LIN {X 0,Y 373.398,Z 423.906,A -85,B 0,C 180,E1 -12851.054,E2 -12851.054} C_VEL
LIN {X 0,Y 371.737,Z 434.746,A -85,B 0,C 180,E1 -12852.96,E2 -12852.96} C_VEL
LIN {X 0,Y 370.406,Z 443.745,A -85,B 0,C 180,E1 -12854.877,E2 -12854.877} C_VEL
LIN {X 0,Y 369.476,Z 451.202,A -85,B 0,C 180,E1 -12856.805,E2 -12856.805} C_VEL
LIN {X 0,Y 368.494,Z 458.177,A -85,B 0,C 180,E1 -12859.005,E2 -12859.005} C_VEL
LIN {X 0,Y 367.969,Z 463.658,A -85,B 0,C 180,E1 -12861.211,E2 -12861.211} C_VEL
LIN {X 0,Y 367.613,Z 468.407,A -85,B 0,C 180,E1 -12863.791,E2 -12863.791} C_VEL
LIN {X 0,Y 367.456,Z 470.707,A -85,B 0,C 180,E1 -12865.612,E2 -12865.612} C_VEL
LIN {X 0,Y 367.353,Z 472.458,A -85,B 0,C 180,E1 -12867.807,E2 -12867.807} C_VEL
LIN {X 0,Y 367.373,Z 473.069,A -85,B 0,C 180,E1 -12870,E2 -12870} C_VEL
LIN {X 0,Y 367.353,Z 472.504,A -85,B 0,C 180,E1 -12872.193,E2 -12872.193} C_VEL
LIN {X 0,Y 367.45,Z 470.815,A -85,B 0,C 180,E1 -12874.388,E2 -12874.388} C_VEL
LIN {X 0,Y 367.559,Z 467.963,A -85,B 0,C 180,E1 -12876.588,E2 -12876.588} C_VEL
LIN {X 0,Y 367.957,Z 463.881,A -85,B 0,C 180,E1 -12878.789,E2 -12878.789} C_VEL
LIN {X 0,Y 368.468,Z 458.469,A -85,B 0,C 180,E1 -12880.996,E2 -12880.996} C_VEL
LIN {X 0,Y 368.933,Z 455.452,A -85,B 0,C 180,E1 -12882.017,E2 -12882.017} C_VEL
LIN {X 0,Y 368.664,Z 452.923,A -85,B 0,C 180,E1 -12882.844,E2 -12882.844} C_VEL
LIN {X 0,Y 366.408,Z 448.547,A -85,B 0,C 180,E1 -12884.185,E2 -12884.185} C_VEL
LIN {X 0,Y 364.21,Z 443.754,A -85,B 0,C 180,E1 -12885.503,E2 -12885.503} C_VEL
LIN {X 0,Y 364.039,Z 440.47,A -85,B 0,C 180,E1 -12886.282,E2 -12886.282} C_VEL
LIN {X 0,Y 365.526,Z 430.926,A -85,B 0,C 180,E1 -12888.206,E2 -12888.206} C_VEL
LIN {X 0,Y 367.184,Z 421.057,A -85,B 0,C 180,E1 -12889.861,E2 -12889.861} C_VEL
LIN {X 0,Y 368.721,Z 410.391,A -85,B 0,C 180,E1 -12891.379,E2 -12891.379} C_VEL
LIN {X 0,Y 370.415,Z 398.934,A -85,B 0,C 180,E1 -12892.742,E2 -12892.742} C_VEL
LIN {X 0,Y 372.09,Z 386.634,A -85,B 0,C 180,E1 -12893.96,E2 -12893.96} C_VEL
LIN {X 0,Y 373.712,Z 373.285,A -85,B 0,C 180,E1 -12895.033,E2 -12895.033} C_VEL
LIN {X 0,Y 375.189,Z 358.112,A -85,B 0,C 180,E1 -12895.993,E2 -12895.993} C_VEL
LIN {X 0,Y 376.337,Z 343.059,A -85,B 0,C 180,E1 -12896.703,E2 -12896.703} C_VEL
LIN {X 0,Y 377.198,Z 327.711,A -85,B 0,C 180,E1 -12897.198,E2 -12897.198} C_VEL
LIN {X 0,Y 380.187,Z 211.478,A -85,B 0,C 180,E1 -12899.438,E2 -12899.438} C_VEL
LIN {X 0,Y 380.388,Z 200.049,A -85,B 0,C 180,E1 -12899.664,E2 -12899.664} C_VEL
LIN {X 0,Y 378.985,Z 193.552,A -85,B 0,C 180,E1 -12899.924,E2 -12899.924} C_VEL
LIN {X 0,Y 370.925,Z 175.178,A -85,B 0,C 180,E1 -12901.05,E2 -12901.05} C_VEL
LIN {X 0,Y 364.955,Z 162.744,A -85,B 0,C 180,E1 -12901.927,E2 -12901.927} C_VEL
LIN {X 0,Y 362.572,Z 153.728,A -85,B 0,C 180,E1 -12904.203,E2 -12904.203} C_VEL
LIN {X 0,Y 361.902,Z 151.154,A -85,B 0,C 180,E1 -12904.951,E2 -12904.951} C_VEL
LIN {X 0,Y 361.843,Z 151.036,A -85,B 0,C 180,E1 -12908.428,E2 -12908.428} C_VEL
LIN {X 0,Y 361.823,Z 151.038,A -85,B 0,C 180,E1 -12912.429,E2 -12912.429} C_VEL
LIN {X 0,Y 361.814,Z 151.039,A -85,B 0,C 180,E1 -12915.948,E2 -12915.948} C_VEL
LIN {X 0,Y 361.81,Z 151.006,A -85,B 0,C 180,E1 -12919.25,E2 -12919.25} C_VEL
LIN {X 0,Y 361.865,Z 151.034,A -85,B 0,C 180,E1 -12922.982,E2 -12922.982} C_VEL
LIN {X 0,Y 361.859,Z 150.996,A -85,B 0,C 180,E1 -12926.631,E2 -12926.631} C_VEL
LIN {X 0,Y 361.849,Z 151.006,A -85,B 0,C 180,E1 -12929.67,E2 -12929.67} C_VEL
LIN {X 0,Y 361.863,Z 151.032,A -85,B 0,C 180,E1 -12933.468,E2 -12933.468} C_VEL
LIN {X 0,Y 361.877,Z 151.031,A -85,B 0,C 180,E1 -12937.144,E2 -12937.144} C_VEL
LIN {X 0,Y 361.885,Z 151.02,A -85,B 0,C 180,E1 -12940.722,E2 -12940.722} C_VEL
LIN {X 0,Y 361.907,Z 151.02,A -85,B 0,C 180,E1 -12944.224,E2 -12944.224} C_VEL
LIN {X 0,Y 362.001,Z 151.007,A -85,B 0,C 180,E1 -12946.528,E2 -12946.528} C_VEL
LIN {X 0,Y 362.002,Z 151.01,A -85,B 0,C 180,E1 -12949.937,E2 -12949.937} C_VEL
LIN {X 0,Y 362.141,Z 150.993,A -85,B 0,C 180,E1 -12953.313,E2 -12953.313} C_VEL
LIN {X 0,Y 362.27,Z 150.965,A -85,B 0,C 180,E1 -12957.776,E2 -12957.776} C_VEL
LIN {X 0,Y 362.382,Z 150.968,A -85,B 0,C 180,E1 -12960,E2 -12960} C_VEL
LIN {X 0,Y 362.274,Z 150.973,A -85,B 0,C 180,E1 -12962.223,E2 -12962.223} C_VEL
LIN {X 0,Y 362.137,Z 150.998,A -85,B 0,C 180,E1 -12966.687,E2 -12966.687} C_VEL
LIN {X 0,Y 362.002,Z 151.001,A -85,B 0,C 180,E1 -12970.063,E2 -12970.063} C_VEL
LIN {X 0,Y 362,Z 151.012,A -85,B 0,C 180,E1 -12973.899,E2 -12973.899} C_VEL
LIN {X 0,Y 361.969,Z 151.02,A -85,B 0,C 180,E1 -12977.938,E2 -12977.938} C_VEL
LIN {X 0,Y 361.862,Z 151.024,A -85,B 0,C 180,E1 -12981.655,E2 -12981.655} C_VEL
LIN {X 0,Y 361.927,Z 151.015,A -85,B 0,C 180,E1 -12985.29,E2 -12985.29} C_VEL
LIN {X 0,Y 361.919,Z 151.025,A -85,B 0,C 180,E1 -12987.778,E2 -12987.778} C_VEL
LIN {X 0,Y 361.847,Z 151.006,A -85,B 0,C 180,E1 -12991.285,E2 -12991.285} C_VEL
LIN {X 0,Y 361.854,Z 150.999,A -85,B 0,C 180,E1 -12994.28,E2 -12994.28} C_VEL
LIN {X 0,Y 361.864,Z 151.034,A -85,B 0,C 180,E1 -12997.223,E2 -12997.223} C_VEL
LIN {X 0,Y 361.835,Z 151.007,A -85,B 0,C 180,E1 -13000.755,E2 -13000.755} C_VEL
LIN {X 0,Y 361.818,Z 151.034,A -85,B 0,C 180,E1 -13004.368,E2 -13004.368} C_VEL
LIN {X 0,Y 361.836,Z 151.03,A -85,B 0,C 180,E1 -13007.568,E2 -13007.568} C_VEL
LIN {X 0,Y 361.869,Z 151.018,A -85,B 0,C 180,E1 -13010.973,E2 -13010.973} C_VEL
LIN {X 0,Y 361.911,Z 151.209,A -85,B 0,C 180,E1 -13013.982,E2 -13013.982} C_VEL
LIN {X 0,Y 365.189,Z 163.283,A -85,B 0,C 180,E1 -13017.076,E2 -13017.076} C_VEL
LIN {X 0,Y 366.498,Z 168.406,A -85,B 0,C 180,E1 -13018.267,E2 -13018.267} C_VEL
LIN {X 0,Y 375.255,Z 187.677,A -85,B 0,C 180,E1 -13019.533,E2 -13019.533} C_VEL
LIN {X 0,Y 377.161,Z 192.668,A -85,B 0,C 180,E1 -13019.811,E2 -13019.811} C_VEL
LIN {X 0,Y 380.221,Z 208.628,A -85,B 0,C 180,E1 -13020.418,E2 -13020.418} C_VEL
LIN {X 0,Y 377.778,Z 309.972,A -85,B 0,C 180,E1 -13022.359,E2 -13022.359} C_VEL
LIN {X 0,Y 377.001,Z 336.104,A -85,B 0,C 180,E1 -13022.899,E2 -13022.899} C_VEL
LIN {X 0,Y 376.013,Z 351.534,A -85,B 0,C 180,E1 -13023.422,E2 -13023.422} C_VEL
LIN {X 0,Y 374.858,Z 365.308,A -85,B 0,C 180,E1 -13024.083,E2 -13024.083} C_VEL
LIN {X 0,Y 373.48,Z 379.072,A -85,B 0,C 180,E1 -13024.953,E2 -13024.953} C_VEL
LIN {X 0,Y 371.868,Z 392.508,A -85,B 0,C 180,E1 -13026.025,E2 -13026.025} C_VEL
LIN {X 0,Y 370.134,Z 404.922,A -85,B 0,C 180,E1 -13027.24,E2 -13027.24} C_VEL
LIN {X 0,Y 368.423,Z 416.478,A -85,B 0,C 180,E1 -13028.603,E2 -13028.603} C_VEL
LIN {X 0,Y 366.803,Z 427.233,A -85,B 0,C 180,E1 -13030.117,E2 -13030.117} C_VEL
LIN {X 0,Y 365.213,Z 437.183,A -85,B 0,C 180,E1 -13031.777,E2 -13031.777} C_VEL
LIN {X 0,Y 363.743,Z 446.916,A -85,B 0,C 180,E1 -13033.73,E2 -13033.73} C_VEL
LIN {X 0,Y 362.496,Z 455.382,A -85,B 0,C 180,E1 -13035.786,E2 -13035.786} C_VEL
LIN {X 0,Y 361.752,Z 461.749,A -85,B 0,C 180,E1 -13037.66,E2 -13037.66} C_VEL
LIN {X 0,Y 360.971,Z 467.946,A -85,B 0,C 180,E1 -13039.908,E2 -13039.908} C_VEL
LIN {X 0,Y 360.582,Z 472.739,A -85,B 0,C 180,E1 -13042.158,E2 -13042.158} C_VEL
LIN {X 0,Y 360.344,Z 476.249,A -85,B 0,C 180,E1 -13044.404,E2 -13044.404} C_VEL
LIN {X 0,Y 360.256,Z 478.558,A -85,B 0,C 180,E1 -13046.645,E2 -13046.645} C_VEL
LIN {X 0,Y 360.245,Z 479.718,A -85,B 0,C 180,E1 -13048.882,E2 -13048.882} C_VEL
LIN {X 0,Y 360.245,Z 479.716,A -85,B 0,C 180,E1 -13051.118,E2 -13051.118} C_VEL
LIN {X 0,Y 360.256,Z 478.546,A -85,B 0,C 180,E1 -13053.355,E2 -13053.355} C_VEL
LIN {X 0,Y 360.348,Z 476.23,A -85,B 0,C 180,E1 -13055.596,E2 -13055.596} C_VEL
LIN {X 0,Y 360.592,Z 472.718,A -85,B 0,C 180,E1 -13057.841,E2 -13057.841} C_VEL
LIN {X 0,Y 360.967,Z 467.92,A -85,B 0,C 180,E1 -13060.092,E2 -13060.092} C_VEL
LIN {X 0,Y 361.746,Z 461.706,A -85,B 0,C 180,E1 -13062.34,E2 -13062.34} C_VEL
LIN {X 0,Y 362.669,Z 453.9,A -85,B 0,C 180,E1 -13064.591,E2 -13064.591} C_VEL
LIN {X 0,Y 363.927,Z 445.6,A -85,B 0,C 180,E1 -13066.55,E2 -13066.55} C_VEL
LIN {X 0,Y 365.473,Z 435.597,A -85,B 0,C 180,E1 -13068.499,E2 -13068.499} C_VEL
LIN {X 0,Y 367.05,Z 424.826,A -85,B 0,C 180,E1 -13070.246,E2 -13070.246} C_VEL
LIN {X 0,Y 368.909,Z 413.17,A -85,B 0,C 180,E1 -13071.808,E2 -13071.808} C_VEL
LIN {X 0,Y 370.812,Z 399.587,A -85,B 0,C 180,E1 -13073.306,E2 -13073.306} C_VEL
LIN {X 0,Y 372.652,Z 385.966,A -85,B 0,C 180,E1 -13074.514,E2 -13074.514} C_VEL
LIN {X 0,Y 374.206,Z 371.977,A -85,B 0,C 180,E1 -13075.509,E2 -13075.509} C_VEL
LIN {X 0,Y 375.479,Z 357.981,A -85,B 0,C 180,E1 -13076.282,E2 -13076.282} C_VEL
LIN {X 0,Y 376.618,Z 342.393,A -85,B 0,C 180,E1 -13076.906,E2 -13076.906} C_VEL
LIN {X 0,Y 377.293,Z 327.061,A -85,B 0,C 180,E1 -13077.303,E2 -13077.303} C_VEL
LIN {X 0,Y 380.19,Z 209.703,A -85,B 0,C 180,E1 -13079.545,E2 -13079.545} C_VEL
LIN {X 0,Y 377.93,Z 196.695,A -85,B 0,C 180,E1 -13080.018,E2 -13080.018} C_VEL
LIN {X 0,Y 376.432,Z 190.399,A -85,B 0,C 180,E1 -13080.285,E2 -13080.285} C_VEL
LIN {X 0,Y 368.092,Z 171.918,A -85,B 0,C 180,E1 -13081.457,E2 -13081.457} C_VEL
LIN {X 0,Y 366.407,Z 168.152,A -85,B 0,C 180,E1 -13081.753,E2 -13081.753} C_VEL
LIN {X 0,Y 363.562,Z 157.181,A -85,B 0,C 180,E1 -13084.432,E2 -13084.432} C_VEL
LIN {X 0,Y 361.894,Z 151.108,A -85,B 0,C 180,E1 -13086.063,E2 -13086.063} C_VEL
LIN {X 0,Y 361.854,Z 151.019,A -85,B 0,C 180,E1 -13089.861,E2 -13089.861} C_VEL
LIN {X 0,Y 361.836,Z 151.022,A -85,B 0,C 180,E1 -13092.829,E2 -13092.829} C_VEL
LIN {X 0,Y 361.819,Z 151.039,A -85,B 0,C 180,E1 -13095.947,E2 -13095.947} C_VEL
LIN {X 0,Y 361.835,Z 151.007,A -85,B 0,C 180,E1 -13099.245,E2 -13099.245} C_VEL
LIN {X 0,Y 361.863,Z 151.034,A -85,B 0,C 180,E1 -13102.777,E2 -13102.777} C_VEL
LIN {X 0,Y 361.853,Z 150.998,A -85,B 0,C 180,E1 -13105.72,E2 -13105.72} C_VEL
LIN {X 0,Y 361.875,Z 151.019,A -85,B 0,C 180,E1 -13109.672,E2 -13109.672} C_VEL
LIN {X 0,Y 361.955,Z 151.01,A -85,B 0,C 180,E1 -13113.475,E2 -13113.475} C_VEL
LIN {X 0,Y 361.891,Z 151.028,A -85,B 0,C 180,E1 -13117.145,E2 -13117.145} C_VEL
LIN {X 0,Y 361.907,Z 151.025,A -85,B 0,C 180,E1 -13120.724,E2 -13120.724} C_VEL
LIN {X 0,Y 361.934,Z 151.018,A -85,B 0,C 180,E1 -13123.066,E2 -13123.066} C_VEL
LIN {X 0,Y 362,Z 151.014,A -85,B 0,C 180,E1 -13126.528,E2 -13126.528} C_VEL
LIN {X 0,Y 362.001,Z 151.001,A -85,B 0,C 180,E1 -13129.937,E2 -13129.937} C_VEL
LIN {X 0,Y 362.137,Z 150.998,A -85,B 0,C 180,E1 -13133.313,E2 -13133.313} C_VEL
LIN {X 0,Y 362.279,Z 150.972,A -85,B 0,C 180,E1 -13137.777,E2 -13137.777} C_VEL
LIN {X 0,Y 362.403,Z 150.965,A -85,B 0,C 180,E1 -13140,E2 -13140} C_VEL
LIN {X 0,Y 362.271,Z 150.965,A -85,B 0,C 180,E1 -13142.224,E2 -13142.224} C_VEL
LIN {X 0,Y 362.141,Z 150.994,A -85,B 0,C 180,E1 -13146.687,E2 -13146.687} C_VEL
LIN {X 0,Y 362.001,Z 151.009,A -85,B 0,C 180,E1 -13150.063,E2 -13150.063} C_VEL
LIN {X 0,Y 362,Z 151.003,A -85,B 0,C 180,E1 -13153.899,E2 -13153.899} C_VEL
LIN {X 0,Y 361.928,Z 151.025,A -85,B 0,C 180,E1 -13156.934,E2 -13156.934} C_VEL
LIN {X 0,Y 361.887,Z 151.018,A -85,B 0,C 180,E1 -13160.461,E2 -13160.461} C_VEL
LIN {X 0,Y 361.862,Z 151.026,A -85,B 0,C 180,E1 -13164.101,E2 -13164.101} C_VEL
LIN {X 0,Y 361.841,Z 151.04,A -85,B 0,C 180,E1 -13167.785,E2 -13167.785} C_VEL
LIN {X 0,Y 361.846,Z 150.992,A -85,B 0,C 180,E1 -13171.285,E2 -13171.285} C_VEL
LIN {X 0,Y 361.854,Z 151.011,A -85,B 0,C 180,E1 -13174.281,E2 -13174.281} C_VEL
LIN {X 0,Y 361.861,Z 151.033,A -85,B 0,C 180,E1 -13177.222,E2 -13177.222} C_VEL
LIN {X 0,Y 361.812,Z 151.003,A -85,B 0,C 180,E1 -13180.751,E2 -13180.751} C_VEL
LIN {X 0,Y 361.815,Z 151.038,A -85,B 0,C 180,E1 -13184.369,E2 -13184.369} C_VEL
LIN {X 0,Y 361.826,Z 151.035,A -85,B 0,C 180,E1 -13187.57,E2 -13187.57} C_VEL
LIN {X 0,Y 361.844,Z 151.034,A -85,B 0,C 180,E1 -13191.572,E2 -13191.572} C_VEL
LIN {X 0,Y 361.921,Z 151.113,A -85,B 0,C 180,E1 -13195.136,E2 -13195.136} C_VEL
LIN {X 0,Y 362.737,Z 154.31,A -85,B 0,C 180,E1 -13196.064,E2 -13196.064} C_VEL
LIN {X 0,Y 365.002,Z 162.815,A -85,B 0,C 180,E1 -13198.195,E2 -13198.195} C_VEL
LIN {X 0,Y 374.821,Z 183.627,A -85,B 0,C 180,E1 -13199.6,E2 -13199.6} C_VEL
LIN {X 0,Y 379.252,Z 194.366,A -85,B 0,C 180,E1 -13200.224,E2 -13200.224} C_VEL
LIN {X 0,Y 380.41,Z 201.067,A -85,B 0,C 180,E1 -13200.466,E2 -13200.466} C_VEL
LIN {X 0,Y 377.588,Z 313.354,A -85,B 0,C 180,E1 -13202.607,E2 -13202.607} C_VEL
LIN {X 0,Y 376.944,Z 332.564,A -85,B 0,C 180,E1 -13203.044,E2 -13203.044} C_VEL
LIN {X 0,Y 375.949,Z 347.72,A -85,B 0,C 180,E1 -13203.598,E2 -13203.598} C_VEL
LIN {X 0,Y 374.794,Z 362.411,A -85,B 0,C 180,E1 -13204.363,E2 -13204.363} C_VEL
LIN {X 0,Y 373.413,Z 375.563,A -85,B 0,C 180,E1 -13205.243,E2 -13205.243} C_VEL
LIN {X 0,Y 371.763,Z 388.509,A -85,B 0,C 180,E1 -13206.314,E2 -13206.314} C_VEL
LIN {X 0,Y 369.97,Z 401.744,A -85,B 0,C 180,E1 -13207.671,E2 -13207.671} C_VEL
LIN {X 0,Y 368.388,Z 412.361,A -85,B 0,C 180,E1 -13208.975,E2 -13208.975} C_VEL
LIN {X 0,Y 366.673,Z 423.976,A -85,B 0,C 180,E1 -13210.693,E2 -13210.693} C_VEL
LIN {X 0,Y 364.905,Z 434.816,A -85,B 0,C 180,E1 -13212.631,E2 -13212.631} C_VEL
LIN {X 0,Y 363.485,Z 443.814,A -85,B 0,C 180,E1 -13214.582,E2 -13214.582} C_VEL
LIN {X 0,Y 362.489,Z 451.271,A -85,B 0,C 180,E1 -13216.546,E2 -13216.546} C_VEL
LIN {X 0,Y 361.482,Z 458.245,A -85,B 0,C 180,E1 -13218.789,E2 -13218.789} C_VEL
LIN {X 0,Y 360.908,Z 463.726,A -85,B 0,C 180,E1 -13221.038,E2 -13221.038} C_VEL
LIN {X 0,Y 360.51,Z 467.865,A -85,B 0,C 180,E1 -13223.283,E2 -13223.283} C_VEL
LIN {X 0,Y 360.368,Z 470.774,A -85,B 0,C 180,E1 -13225.526,E2 -13225.526} C_VEL
LIN {X 0,Y 360.258,Z 472.524,A -85,B 0,C 180,E1 -13227.764,E2 -13227.764} C_VEL
LIN {X 0,Y 360.273,Z 473.135,A -85,B 0,C 180,E1 -13230,E2 -13230} C_VEL
LIN {X 0,Y 360.258,Z 472.57,A -85,B 0,C 180,E1 -13232.236,E2 -13232.236} C_VEL
LIN {X 0,Y 360.361,Z 470.88,A -85,B 0,C 180,E1 -13234.474,E2 -13234.474} C_VEL
LIN {X 0,Y 360.491,Z 468.029,A -85,B 0,C 180,E1 -13236.718,E2 -13236.718} C_VEL
LIN {X 0,Y 360.892,Z 463.946,A -85,B 0,C 180,E1 -13238.963,E2 -13238.963} C_VEL
LIN {X 0,Y 361.457,Z 458.535,A -85,B 0,C 180,E1 -13241.212,E2 -13241.212} C_VEL
LIN {X 0,Y 362.199,Z 453.482,A -85,B 0,C 180,E1 -13242.894,E2 -13242.894} C_VEL
LIN {X 0,Y 363.091,Z 446.455,A -85,B 0,C 180,E1 -13244.861,E2 -13244.861} C_VEL
LIN {X 0,Y 364.039,Z 440.47,A -85,B 0,C 180,E1 -13246.282,E2 -13246.282} C_VEL
LIN {X 0,Y 363.957,Z 437.104,A -85,B 0,C 180,E1 -13247.045,E2 -13247.045} C_VEL
LIN {X 0,Y 362.185,Z 431.465,A -85,B 0,C 180,E1 -13248.298,E2 -13248.298} C_VEL
LIN {X 0,Y 360.448,Z 425.436,A -85,B 0,C 180,E1 -13249.512,E2 -13249.512} C_VEL
LIN {X 0,Y 360.414,Z 421.409,A -85,B 0,C 180,E1 -13250.202,E2 -13250.202} C_VEL
LIN {X 0,Y 361.914,Z 411.522,A -85,B 0,C 180,E1 -13251.652,E2 -13251.652} C_VEL
LIN {X 0,Y 363.865,Z 398.996,A -85,B 0,C 180,E1 -13253.175,E2 -13253.175} C_VEL
LIN {X 0,Y 365.582,Z 386.695,A -85,B 0,C 180,E1 -13254.414,E2 -13254.414} C_VEL
LIN {X 0,Y 367.267,Z 373.345,A -85,B 0,C 180,E1 -13255.503,E2 -13255.503} C_VEL
LIN {X 0,Y 368.764,Z 358.764,A -85,B 0,C 180,E1 -13256.444,E2 -13256.444} C_VEL
LIN {X 0,Y 369.949,Z 343.934,A -85,B 0,C 180,E1 -13257.163,E2 -13257.163} C_VEL
LIN {X 0,Y 370.917,Z 327.757,A -85,B 0,C 180,E1 -13257.698,E2 -13257.698} C_VEL
LIN {X 0,Y 373.772,Z 221.488,A -85,B 0,C 180,E1 -13259.778,E2 -13259.778} C_VEL
LIN {X 0,Y 374.215,Z 201.101,A -85,B 0,C 180,E1 -13260.181,E2 -13260.181} C_VEL
LIN {X 0,Y 373.022,Z 195.908,A -85,B 0,C 180,E1 -13260.402,E2 -13260.402} C_VEL
LIN {X 0,Y 364.42,Z 176.546,A -85,B 0,C 180,E1 -13261.638,E2 -13261.638} C_VEL
LIN {X 0,Y 357.7,Z 162.698,A -85,B 0,C 180,E1 -13262.666,E2 -13262.666} C_VEL
LIN {X 0,Y 354.93,Z 152.51,A -85,B 0,C 180,E1 -13265.365,E2 -13265.365} C_VEL
LIN {X 0,Y 354.819,Z 151.924,A -85,B 0,C 180,E1 -13265.698,E2 -13265.698} C_VEL
LIN {X 0,Y 354.769,Z 151.904,A -85,B 0,C 180,E1 -13269.412,E2 -13269.412} C_VEL
LIN {X 0,Y 354.781,Z 151.907,A -85,B 0,C 180,E1 -13272.866,E2 -13272.866} C_VEL
LIN {X 0,Y 354.763,Z 151.917,A -85,B 0,C 180,E1 -13276.103,E2 -13276.103} C_VEL
LIN {X 0,Y 354.763,Z 151.883,A -85,B 0,C 180,E1 -13279.175,E2 -13279.175} C_VEL
LIN {X 0,Y 354.801,Z 151.905,A -85,B 0,C 180,E1 -13282.404,E2 -13282.404} C_VEL
LIN {X 0,Y 354.813,Z 151.906,A -85,B 0,C 180,E1 -13284.941,E2 -13284.941} C_VEL
LIN {X 0,Y 354.79,Z 151.865,A -85,B 0,C 180,E1 -13288.406,E2 -13288.406} C_VEL
LIN {X 0,Y 354.8,Z 151.911,A -85,B 0,C 180,E1 -13291.614,E2 -13291.614} C_VEL
LIN {X 0,Y 354.805,Z 151.901,A -85,B 0,C 180,E1 -13295.42,E2 -13295.42} C_VEL
LIN {X 0,Y 354.828,Z 151.902,A -85,B 0,C 180,E1 -13299.113,E2 -13299.113} C_VEL
LIN {X 0,Y 354.862,Z 151.905,A -85,B 0,C 180,E1 -13302.718,E2 -13302.718} C_VEL
LIN {X 0,Y 354.942,Z 151.882,A -85,B 0,C 180,E1 -13306.255,E2 -13306.255} C_VEL
LIN {X 0,Y 354.958,Z 151.889,A -85,B 0,C 180,E1 -13309.735,E2 -13309.735} C_VEL
LIN {X 0,Y 355.104,Z 151.869,A -85,B 0,C 180,E1 -13313.18,E2 -13313.18} C_VEL
LIN {X 0,Y 355.232,Z 151.841,A -85,B 0,C 180,E1 -13317.732,E2 -13317.732} C_VEL
LIN {X 0,Y 355.333,Z 151.846,A -85,B 0,C 180,E1 -13320,E2 -13320} C_VEL
LIN {X 0,Y 355.236,Z 151.849,A -85,B 0,C 180,E1 -13322.268,E2 -13322.268} C_VEL
LIN {X 0,Y 355.1,Z 151.875,A -85,B 0,C 180,E1 -13326.82,E2 -13326.82} C_VEL
LIN {X 0,Y 354.958,Z 151.879,A -85,B 0,C 180,E1 -13330.265,E2 -13330.265} C_VEL
LIN {X 0,Y 354.945,Z 151.89,A -85,B 0,C 180,E1 -13334.019,E2 -13334.019} C_VEL
LIN {X 0,Y 354.924,Z 151.898,A -85,B 0,C 180,E1 -13338.108,E2 -13338.108} C_VEL
LIN {X 0,Y 354.817,Z 151.904,A -85,B 0,C 180,E1 -13342.107,E2 -13342.107} C_VEL
LIN {X 0,Y 354.899,Z 151.888,A -85,B 0,C 180,E1 -13345.827,E2 -13345.827} C_VEL
LIN {X 0,Y 354.855,Z 151.903,A -85,B 0,C 180,E1 -13349.678,E2 -13349.678} C_VEL
LIN {X 0,Y 354.807,Z 151.867,A -85,B 0,C 180,E1 -13353.702,E2 -13353.702} C_VEL
LIN {X 0,Y 354.798,Z 151.913,A -85,B 0,C 180,E1 -13356.459,E2 -13356.459} C_VEL
LIN {X 0,Y 354.825,Z 151.884,A -85,B 0,C 180,E1 -13359.423,E2 -13359.423} C_VEL
LIN {X 0,Y 354.789,Z 151.915,A -85,B 0,C 180,E1 -13362.867,E2 -13362.867} C_VEL
LIN {X 0,Y 354.767,Z 151.894,A -85,B 0,C 180,E1 -13366.103,E2 -13366.103} C_VEL
LIN {X 0,Y 354.788,Z 151.909,A -85,B 0,C 180,E1 -13369.179,E2 -13369.179} C_VEL
LIN {X 0,Y 354.83,Z 151.907,A -85,B 0,C 180,E1 -13372.835,E2 -13372.835} C_VEL
LIN {X 0,Y 354.875,Z 152.086,A -85,B 0,C 180,E1 -13373.373,E2 -13373.373} C_VEL
LIN {X 0,Y 358.335,Z 164.655,A -85,B 0,C 180,E1 -13376.69,E2 -13376.69} C_VEL
LIN {X 0,Y 359.265,Z 168.47,A -85,B 0,C 180,E1 -13377.558,E2 -13377.558} C_VEL
LIN {X 0,Y 368.825,Z 188.945,A -85,B 0,C 180,E1 -13378.973,E2 -13378.973} C_VEL
LIN {X 0,Y 371.273,Z 195.231,A -85,B 0,C 180,E1 -13379.338,E2 -13379.338} C_VEL
LIN {X 0,Y 374.05,Z 209.806,A -85,B 0,C 180,E1 -13379.907,E2 -13379.907} C_VEL
LIN {X 0,Y 371.509,Z 309.926,A -85,B 0,C 180,E1 -13381.852,E2 -13381.852} C_VEL
LIN {X 0,Y 370.693,Z 336.05,A -85,B 0,C 180,E1 -13382.399,E2 -13382.399} C_VEL
LIN {X 0,Y 369.688,Z 351.477,A -85,B 0,C 180,E1 -13382.931,E2 -13382.931} C_VEL
LIN {X 0,Y 368.488,Z 365.248,A -85,B 0,C 180,E1 -13383.601,E2 -13383.601} C_VEL
LIN {X 0,Y 367,Z 379.419,A -85,B 0,C 180,E1 -13384.512,E2 -13384.512} C_VEL
LIN {X 0,Y 365.162,Z 393.954,A -85,B 0,C 180,E1 -13385.708,E2 -13385.708} C_VEL
LIN {X 0,Y 363.377,Z 406.151,A -85,B 0,C 180,E1 -13386.943,E2 -13386.943} C_VEL
LIN {X 0,Y 361.452,Z 418.557,A -85,B 0,C 180,E1 -13388.469,E2 -13388.469} C_VEL
LIN {X 0,Y 359.769,Z 429.213,A -85,B 0,C 180,E1 -13390.053,E2 -13390.053} C_VEL
LIN {X 0,Y 358.139,Z 438.605,A -85,B 0,C 180,E1 -13391.701,E2 -13391.701} C_VEL
LIN {X 0,Y 356.65,Z 448.085,A -85,B 0,C 180,E1 -13393.692,E2 -13393.692} C_VEL
LIN {X 0,Y 355.368,Z 456.653,A -85,B 0,C 180,E1 -13395.882,E2 -13395.882} C_VEL
LIN {X 0,Y 354.541,Z 463.352,A -85,B 0,C 180,E1 -13397.987,E2 -13397.987} C_VEL
LIN {X 0,Y 353.801,Z 469.198,A -85,B 0,C 180,E1 -13400.279,E2 -13400.279} C_VEL
LIN {X 0,Y 353.511,Z 472.673,A -85,B 0,C 180,E1 -13402,E2 -13402} C_VEL
LIN {X 0,Y 353.28,Z 476.184,A -85,B 0,C 180,E1 -13404.291,E2 -13404.291} C_VEL
LIN {X 0,Y 353.179,Z 478.492,A -85,B 0,C 180,E1 -13406.577,E2 -13406.577} C_VEL
LIN {X 0,Y 353.144,Z 479.652,A -85,B 0,C 180,E1 -13408.86,E2 -13408.86} C_VEL
LIN {X 0,Y 353.144,Z 479.65,A -85,B 0,C 180,E1 -13411.14,E2 -13411.14} C_VEL
LIN {X 0,Y 353.179,Z 478.479,A -85,B 0,C 180,E1 -13413.422,E2 -13413.422} C_VEL
LIN {X 0,Y 353.292,Z 475.876,A -85,B 0,C 180,E1 -13415.934,E2 -13415.934} C_VEL
LIN {X 0,Y 353.595,Z 471.582,A -85,B 0,C 180,E1 -13418.573,E2 -13418.573} C_VEL
LIN {X 0,Y 354.051,Z 466.422,A -85,B 0,C 180,E1 -13420.87,E2 -13420.87} C_VEL
LIN {X 0,Y 354.943,Z 459.823,A -85,B 0,C 180,E1 -13423.162,E2 -13423.162} C_VEL
LIN {X 0,Y 355.916,Z 452.714,A -85,B 0,C 180,E1 -13425.167,E2 -13425.167} C_VEL
LIN {X 0,Y 357.254,Z 444.175,A -85,B 0,C 180,E1 -13427.163,E2 -13427.163} C_VEL
LIN {X 0,Y 358.711,Z 435.528,A -85,B 0,C 180,E1 -13428.861,E2 -13428.861} C_VEL
LIN {X 0,Y 360.248,Z 425.295,A -85,B 0,C 180,E1 -13430.558,E2 -13430.558} C_VEL
LIN {X 0,Y 362.289,Z 413.1,A -85,B 0,C 180,E1 -13432.227,E2 -13432.227} C_VEL
LIN {X 0,Y 364.287,Z 399.517,A -85,B 0,C 180,E1 -13433.749,E2 -13433.749} C_VEL
LIN {X 0,Y 366.2,Z 385.895,A -85,B 0,C 180,E1 -13434.975,E2 -13434.975} C_VEL
LIN {X 0,Y 367.833,Z 371.736,A -85,B 0,C 180,E1 -13435.996,E2 -13435.996} C_VEL
LIN {X 0,Y 369.111,Z 357.907,A -85,B 0,C 180,E1 -13436.771,E2 -13436.771} C_VEL
LIN {X 0,Y 370.315,Z 342.316,A -85,B 0,C 180,E1 -13437.402,E2 -13437.402} C_VEL
LIN {X 0,Y 371.01,Z 326.978,A -85,B 0,C 180,E1 -13437.805,E2 -13437.805} C_VEL
LIN {X 0,Y 373.828,Z 217.019,A -85,B 0,C 180,E1 -13439.939,E2 -13439.939} C_VEL
LIN {X 0,Y 373.924,Z 209.275,A -85,B 0,C 180,E1 -13440.098,E2 -13440.098} C_VEL
LIN {X 0,Y 370.839,Z 193.776,A -85,B 0,C 180,E1 -13440.715,E2 -13440.715} C_VEL
LIN {X 0,Y 362.754,Z 175.77,A -85,B 0,C 180,E1 -13441.884,E2 -13441.884} C_VEL
LIN {X 0,Y 359.171,Z 168.123,A -85,B 0,C 180,E1 -13442.462,E2 -13442.462} C_VEL
LIN {X 0,Y 356.042,Z 156.407,A -85,B 0,C 180,E1 -13445.428,E2 -13445.428} C_VEL
LIN {X 0,Y 354.848,Z 151.967,A -85,B 0,C 180,E1 -13446.674,E2 -13446.674} C_VEL
LIN {X 0,Y 354.824,Z 151.893,A -85,B 0,C 180,E1 -13449.424,E2 -13449.424} C_VEL
LIN {X 0,Y 354.788,Z 151.899,A -85,B 0,C 180,E1 -13452.867,E2 -13452.867} C_VEL
LIN {X 0,Y 354.767,Z 151.919,A -85,B 0,C 180,E1 -13456.104,E2 -13456.104} C_VEL
LIN {X 0,Y 354.787,Z 151.884,A -85,B 0,C 180,E1 -13459.179,E2 -13459.179} C_VEL
LIN {X 0,Y 354.807,Z 151.913,A -85,B 0,C 180,E1 -13462.403,E2 -13462.403} C_VEL
LIN {X 0,Y 354.811,Z 151.888,A -85,B 0,C 180,E1 -13464.941,E2 -13464.941} C_VEL
LIN {X 0,Y 354.793,Z 151.878,A -85,B 0,C 180,E1 -13468.406,E2 -13468.406} C_VEL
LIN {X 0,Y 354.852,Z 151.908,A -85,B 0,C 180,E1 -13471.619,E2 -13471.619} C_VEL
LIN {X 0,Y 354.9,Z 151.888,A -85,B 0,C 180,E1 -13474.173,E2 -13474.173} C_VEL
LIN {X 0,Y 354.836,Z 151.901,A -85,B 0,C 180,E1 -13477.894,E2 -13477.894} C_VEL
LIN {X 0,Y 354.923,Z 151.898,A -85,B 0,C 180,E1 -13481.892,E2 -13481.892} C_VEL
LIN {X 0,Y 354.944,Z 151.891,A -85,B 0,C 180,E1 -13485.981,E2 -13485.981} C_VEL
LIN {X 0,Y 354.957,Z 151.879,A -85,B 0,C 180,E1 -13489.735,E2 -13489.735} C_VEL
LIN {X 0,Y 355.1,Z 151.876,A -85,B 0,C 180,E1 -13493.18,E2 -13493.18} C_VEL
LIN {X 0,Y 355.242,Z 151.848,A -85,B 0,C 180,E1 -13497.732,E2 -13497.732} C_VEL
LIN {X 0,Y 355.353,Z 151.843,A -85,B 0,C 180,E1 -13500,E2 -13500} C_VEL
LIN {X 0,Y 355.234,Z 151.841,A -85,B 0,C 180,E1 -13502.268,E2 -13502.268} C_VEL
LIN {X 0,Y 355.103,Z 151.869,A -85,B 0,C 180,E1 -13506.82,E2 -13506.82} C_VEL
LIN {X 0,Y 354.957,Z 151.889,A -85,B 0,C 180,E1 -13510.265,E2 -13510.265} C_VEL
LIN {X 0,Y 354.944,Z 151.881,A -85,B 0,C 180,E1 -13514.019,E2 -13514.019} C_VEL
LIN {X 0,Y 354.891,Z 151.9,A -85,B 0,C 180,E1 -13518.092,E2 -13518.092} C_VEL
LIN {X 0,Y 354.815,Z 151.913,A -85,B 0,C 180,E1 -13522.107,E2 -13522.107} C_VEL
LIN {X 0,Y 354.803,Z 151.902,A -85,B 0,C 180,E1 -13525.835,E2 -13525.835} C_VEL
LIN {X 0,Y 354.794,Z 151.898,A -85,B 0,C 180,E1 -13529.684,E2 -13529.684} C_VEL
LIN {X 0,Y 354.785,Z 151.864,A -85,B 0,C 180,E1 -13532.334,E2 -13532.334} C_VEL
LIN {X 0,Y 354.822,Z 151.91,A -85,B 0,C 180,E1 -13535.699,E2 -13535.699} C_VEL
LIN {X 0,Y 354.768,Z 151.881,A -85,B 0,C 180,E1 -13539.413,E2 -13539.413} C_VEL
LIN {X 0,Y 354.786,Z 151.913,A -85,B 0,C 180,E1 -13542.867,E2 -13542.867} C_VEL
LIN {X 0,Y 354.763,Z 151.898,A -85,B 0,C 180,E1 -13546.103,E2 -13546.103} C_VEL
LIN {X 0,Y 354.764,Z 151.91,A -85,B 0,C 180,E1 -13549.176,E2 -13549.176} C_VEL
LIN {X 0,Y 354.8,Z 151.913,A -85,B 0,C 180,E1 -13552.404,E2 -13552.404} C_VEL
LIN {X 0,Y 354.835,Z 152.001,A -85,B 0,C 180,E1 -13554.535,E2 -13554.535} C_VEL
LIN {X 0,Y 355.507,Z 154.522,A -85,B 0,C 180,E1 -13555.307,E2 -13555.307} C_VEL
LIN {X 0,Y 357.768,Z 162.9,A -85,B 0,C 180,E1 -13557.473,E2 -13557.473} C_VEL
LIN {X 0,Y 365.727,Z 179.348,A -85,B 0,C 180,E1 -13558.661,E2 -13558.661} C_VEL
LIN {X 0,Y 373.107,Z 196.191,A -85,B 0,C 180,E1 -13559.72,E2 -13559.72} C_VEL
LIN {X 0,Y 374.201,Z 202.372,A -85,B 0,C 180,E1 -13559.953,E2 -13559.953} C_VEL
LIN {X 0,Y 370.941,Z 326.599,A -85,B 0,C 180,E1 -13562.381,E2 -13562.381} C_VEL
LIN {X 0,Y 370.102,Z 341.502,A -85,B 0,C 180,E1 -13562.849,E2 -13562.849} C_VEL
LIN {X 0,Y 368.996,Z 355.54,A -85,B 0,C 180,E1 -13563.488,E2 -13563.488} C_VEL
LIN {X 0,Y 367.597,Z 370.003,A -85,B 0,C 180,E1 -13564.37,E2 -13564.37} C_VEL
LIN {X 0,Y 365.896,Z 384.007,A -85,B 0,C 180,E1 -13565.458,E2 -13565.458} C_VEL
LIN {X 0,Y 364.16,Z 396.81,A -85,B 0,C 180,E1 -13566.694,E2 -13566.694} C_VEL
LIN {X 0,Y 362.104,Z 409.711,A -85,B 0,C 180,E1 -13568.211,E2 -13568.211} C_VEL
LIN {X 0,Y 360.493,Z 420.494,A -85,B 0,C 180,E1 -13569.754,E2 -13569.754} C_VEL
LIN {X 0,Y 358.816,Z 430.466,A -85,B 0,C 180,E1 -13571.441,E2 -13571.441} C_VEL
LIN {X 0,Y 357.217,Z 440.206,A -85,B 0,C 180,E1 -13573.425,E2 -13573.425} C_VEL
LIN {X 0,Y 355.915,Z 448.149,A -85,B 0,C 180,E1 -13575.369,E2 -13575.369} C_VEL
LIN {X 0,Y 355.028,Z 455.024,A -85,B 0,C 180,E1 -13577.423,E2 -13577.423} C_VEL
LIN {X 0,Y 354.145,Z 461.23,A -85,B 0,C 180,E1 -13579.712,E2 -13579.712} C_VEL
LIN {X 0,Y 353.621,Z 466.023,A -85,B 0,C 180,E1 -13582.003,E2 -13582.003} C_VEL
LIN {X 0,Y 353.348,Z 469.535,A -85,B 0,C 180,E1 -13584.293,E2 -13584.293} C_VEL
LIN {X 0,Y 353.217,Z 471.858,A -85,B 0,C 180,E1 -13586.578,E2 -13586.578} C_VEL
LIN {X 0,Y 353.155,Z 473.044,A -85,B 0,C 180,E1 -13588.86,E2 -13588.86} C_VEL
LIN {X 0,Y 353.156,Z 473.059,A -85,B 0,C 180,E1 -13591.14,E2 -13591.14} C_VEL
LIN {X 0,Y 353.216,Z 471.933,A -85,B 0,C 180,E1 -13593.422,E2 -13593.422} C_VEL
LIN {X 0,Y 353.33,Z 469.67,A -85,B 0,C 180,E1 -13595.708,E2 -13595.708} C_VEL
LIN {X 0,Y 353.612,Z 466.212,A -85,B 0,C 180,E1 -13597.997,E2 -13597.997} C_VEL
LIN {X 0,Y 354.121,Z 461.48,A -85,B 0,C 180,E1 -13600.289,E2 -13600.289} C_VEL
LIN {X 0,Y 354.982,Z 455.35,A -85,B 0,C 180,E1 -13602.579,E2 -13602.579} C_VEL
LIN {X 0,Y 356.016,Z 447.634,A -85,B 0,C 180,E1 -13604.87,E2 -13604.87} C_VEL
LIN {X 0,Y 357.378,Z 439.407,A -85,B 0,C 180,E1 -13606.862,E2 -13606.862} C_VEL
LIN {X 0,Y 358.986,Z 429.499,A -85,B 0,C 180,E1 -13608.846,E2 -13608.846} C_VEL
LIN {X 0,Y 360.414,Z 421.409,A -85,B 0,C 180,E1 -13610.202,E2 -13610.202} C_VEL
LIN {X 0,Y 360.406,Z 417.312,A -85,B 0,C 180,E1 -13610.877,E2 -13610.877} C_VEL
LIN {X 0,Y 358.814,Z 410.547,A -85,B 0,C 180,E1 -13612.008,E2 -13612.008} C_VEL
LIN {X 0,Y 357.287,Z 403.442,A -85,B 0,C 180,E1 -13613.082,E2 -13613.082} C_VEL
LIN {X 0,Y 357.359,Z 398.766,A -85,B 0,C 180,E1 -13613.657,E2 -13613.657} C_VEL
LIN {X 0,Y 359.122,Z 386.756,A -85,B 0,C 180,E1 -13614.882,E2 -13614.882} C_VEL
LIN {X 0,Y 360.859,Z 373.405,A -85,B 0,C 180,E1 -13615.99,E2 -13615.99} C_VEL
LIN {X 0,Y 362.436,Z 358.661,A -85,B 0,C 180,E1 -13616.953,E2 -13616.953} C_VEL
LIN {X 0,Y 363.664,Z 343.989,A -85,B 0,C 180,E1 -13617.673,E2 -13617.673} C_VEL
LIN {X 0,Y 364.652,Z 327.804,A -85,B 0,C 180,E1 -13618.216,E2 -13618.216} C_VEL
LIN {X 0,Y 367.605,Z 222.873,A -85,B 0,C 180,E1 -13620.299,E2 -13620.299} C_VEL
LIN {X 0,Y 368.091,Z 202.193,A -85,B 0,C 180,E1 -13620.714,E2 -13620.714} C_VEL
LIN {X 0,Y 367.102,Z 198.532,A -85,B 0,C 180,E1 -13620.888,E2 -13620.888} C_VEL
LIN {X 0,Y 360.17,Z 182.646,A -85,B 0,C 180,E1 -13621.916,E2 -13621.916} C_VEL
LIN {X 0,Y 351.983,Z 165.915,A -85,B 0,C 180,E1 -13623.149,E2 -13623.149} C_VEL
LIN {X 0,Y 350.497,Z 162.61,A -85,B 0,C 180,E1 -13623.445,E2 -13623.445} C_VEL
LIN {X 0,Y 347.827,Z 153.141,A -85,B 0,C 180,E1 -13626.078,E2 -13626.078} C_VEL
LIN {X 0,Y 347.773,Z 152.81,A -85,B 0,C 180,E1 -13626.299,E2 -13626.299} C_VEL
LIN {X 0,Y 347.701,Z 152.782,A -85,B 0,C 180,E1 -13629.818,E2 -13629.818} C_VEL
LIN {X 0,Y 347.721,Z 152.778,A -85,B 0,C 180,E1 -13633.409,E2 -13633.409} C_VEL
LIN {X 0,Y 347.723,Z 152.799,A -85,B 0,C 180,E1 -13636.687,E2 -13636.687} C_VEL
LIN {X 0,Y 347.701,Z 152.757,A -85,B 0,C 180,E1 -13640.182,E2 -13640.182} C_VEL
LIN {X 0,Y 347.757,Z 152.786,A -85,B 0,C 180,E1 -13642.678,E2 -13642.678} C_VEL
LIN {X 0,Y 347.75,Z 152.764,A -85,B 0,C 180,E1 -13645.956,E2 -13645.956} C_VEL
LIN {X 0,Y 347.736,Z 152.76,A -85,B 0,C 180,E1 -13649.651,E2 -13649.651} C_VEL
LIN {X 0,Y 347.744,Z 152.789,A -85,B 0,C 180,E1 -13653.6,E2 -13653.6} C_VEL
LIN {X 0,Y 347.753,Z 152.784,A -85,B 0,C 180,E1 -13656.159,E2 -13656.159} C_VEL
LIN {X 0,Y 347.8,Z 152.771,A -85,B 0,C 180,E1 -13659.908,E2 -13659.908} C_VEL
LIN {X 0,Y 347.835,Z 152.783,A -85,B 0,C 180,E1 -13662.357,E2 -13662.357} C_VEL
LIN {X 0,Y 347.9,Z 152.757,A -85,B 0,C 180,E1 -13665.971,E2 -13665.971} C_VEL
LIN {X 0,Y 347.899,Z 152.772,A -85,B 0,C 180,E1 -13669.525,E2 -13669.525} C_VEL
LIN {X 0,Y 348.068,Z 152.745,A -85,B 0,C 180,E1 -13673.041,E2 -13673.041} C_VEL
LIN {X 0,Y 348.194,Z 152.717,A -85,B 0,C 180,E1 -13677.686,E2 -13677.686} C_VEL
LIN {X 0,Y 348.285,Z 152.724,A -85,B 0,C 180,E1 -13680,E2 -13680} C_VEL
LIN {X 0,Y 348.198,Z 152.725,A -85,B 0,C 180,E1 -13682.313,E2 -13682.313} C_VEL
LIN {X 0,Y 348.065,Z 152.753,A -85,B 0,C 180,E1 -13686.958,E2 -13686.958} C_VEL
LIN {X 0,Y 347.898,Z 152.76,A -85,B 0,C 180,E1 -13690.475,E2 -13690.475} C_VEL
LIN {X 0,Y 347.9,Z 152.768,A -85,B 0,C 180,E1 -13694.15,E2 -13694.15} C_VEL
LIN {X 0,Y 347.892,Z 152.774,A -85,B 0,C 180,E1 -13698.29,E2 -13698.29} C_VEL
LIN {X 0,Y 347.769,Z 152.778,A -85,B 0,C 180,E1 -13701.626,E2 -13701.626} C_VEL
LIN {X 0,Y 347.812,Z 152.774,A -85,B 0,C 180,E1 -13705.108,E2 -13705.108} C_VEL
LIN {X 0,Y 347.812,Z 152.783,A -85,B 0,C 180,E1 -13707.694,E2 -13707.694} C_VEL
LIN {X 0,Y 347.765,Z 152.774,A -85,B 0,C 180,E1 -13710.346,E2 -13710.346} C_VEL
LIN {X 0,Y 347.745,Z 152.757,A -85,B 0,C 180,E1 -13714.464,E2 -13714.464} C_VEL
LIN {X 0,Y 347.774,Z 152.784,A -85,B 0,C 180,E1 -13717.988,E2 -13717.988} C_VEL
LIN {X 0,Y 347.751,Z 152.772,A -85,B 0,C 180,E1 -13721.83,E2 -13721.83} C_VEL
LIN {X 0,Y 347.706,Z 152.781,A -85,B 0,C 180,E1 -13725.027,E2 -13725.027} C_VEL
LIN {X 0,Y 347.751,Z 152.795,A -85,B 0,C 180,E1 -13728.397,E2 -13728.397} C_VEL
LIN {X 0,Y 347.776,Z 152.786,A -85,B 0,C 180,E1 -13732.011,E2 -13732.011} C_VEL
LIN {X 0,Y 347.84,Z 153.062,A -85,B 0,C 180,E1 -13732.772,E2 -13732.772} C_VEL
LIN {X 0,Y 351.424,Z 165.987,A -85,B 0,C 180,E1 -13736.272,E2 -13736.272} C_VEL
LIN {X 0,Y 352.07,Z 168.372,A -85,B 0,C 180,E1 -13736.809,E2 -13736.809} C_VEL
LIN {X 0,Y 361.506,Z 188.413,A -85,B 0,C 180,E1 -13738.262,E2 -13738.262} C_VEL
LIN {X 0,Y 365.427,Z 197.757,A -85,B 0,C 180,E1 -13738.851,E2 -13738.851} C_VEL
LIN {X 0,Y 367.908,Z 211.014,A -85,B 0,C 180,E1 -13739.379,E2 -13739.379} C_VEL
LIN {X 0,Y 365.172,Z 311.669,A -85,B 0,C 180,E1 -13741.358,E2 -13741.358} C_VEL
LIN {X 0,Y 364.432,Z 335.997,A -85,B 0,C 180,E1 -13741.883,E2 -13741.883} C_VEL
LIN {X 0,Y 363.368,Z 351.57,A -85,B 0,C 180,E1 -13742.428,E2 -13742.428} C_VEL
LIN {X 0,Y 362.054,Z 366.05,A -85,B 0,C 180,E1 -13743.154,E2 -13743.154} C_VEL
LIN {X 0,Y 360.553,Z 379.72,A -85,B 0,C 180,E1 -13744.054,E2 -13744.054} C_VEL
LIN {X 0,Y 358.691,Z 393.892,A -85,B 0,C 180,E1 -13745.24,E2 -13745.24} C_VEL
LIN {X 0,Y 356.799,Z 406.088,A -85,B 0,C 180,E1 -13746.492,E2 -13746.492} C_VEL
LIN {X 0,Y 354.802,Z 418.492,A -85,B 0,C 180,E1 -13748.045,E2 -13748.045} C_VEL
LIN {X 0,Y 353.001,Z 429.499,A -85,B 0,C 180,E1 -13749.713,E2 -13749.713} C_VEL
LIN {X 0,Y 351.116,Z 440.028,A -85,B 0,C 180,E1 -13751.624,E2 -13751.624} C_VEL
LIN {X 0,Y 349.576,Z 449.253,A -85,B 0,C 180,E1 -13753.653,E2 -13753.653} C_VEL
LIN {X 0,Y 348.252,Z 457.936,A -85,B 0,C 180,E1 -13755.985,E2 -13755.985} C_VEL
LIN {X 0,Y 347.28,Z 464.902,A -85,B 0,C 180,E1 -13758.324,E2 -13758.324} C_VEL
LIN {X 0,Y 346.638,Z 470.377,A -85,B 0,C 180,E1 -13760.665,E2 -13760.665} C_VEL
LIN {X 0,Y 346.316,Z 474.517,A -85,B 0,C 180,E1 -13763.006,E2 -13763.006} C_VEL
LIN {X 0,Y 346.129,Z 477.418,A -85,B 0,C 180,E1 -13765.341,E2 -13765.341} C_VEL
LIN {X 0,Y 346.04,Z 479.147,A -85,B 0,C 180,E1 -13767.672,E2 -13767.672} C_VEL
LIN {X 0,Y 346.073,Z 479.739,A -85,B 0,C 180,E1 -13770,E2 -13770} C_VEL
LIN {X 0,Y 346.04,Z 479.139,A -85,B 0,C 180,E1 -13772.328,E2 -13772.328} C_VEL
LIN {X 0,Y 346.13,Z 477.4,A -85,B 0,C 180,E1 -13774.659,E2 -13774.659} C_VEL
LIN {X 0,Y 346.318,Z 474.494,A -85,B 0,C 180,E1 -13776.994,E2 -13776.994} C_VEL
LIN {X 0,Y 346.633,Z 470.351,A -85,B 0,C 180,E1 -13779.335,E2 -13779.335} C_VEL
LIN {X 0,Y 347.275,Z 464.863,A -85,B 0,C 180,E1 -13781.676,E2 -13781.676} C_VEL
LIN {X 0,Y 348.213,Z 457.879,A -85,B 0,C 180,E1 -13784.016,E2 -13784.016} C_VEL
LIN {X 0,Y 349.577,Z 449.187,A -85,B 0,C 180,E1 -13786.347,E2 -13786.347} C_VEL
LIN {X 0,Y 351.086,Z 439.952,A -85,B 0,C 180,E1 -13788.378,E2 -13788.378} C_VEL
LIN {X 0,Y 352.929,Z 429.595,A -85,B 0,C 180,E1 -13790.258,E2 -13790.258} C_VEL
LIN {X 0,Y 354.783,Z 418.383,A -85,B 0,C 180,E1 -13791.956,E2 -13791.956} C_VEL
LIN {X 0,Y 356.806,Z 405.959,A -85,B 0,C 180,E1 -13793.507,E2 -13793.507} C_VEL
LIN {X 0,Y 358.826,Z 392.207,A -85,B 0,C 180,E1 -13794.904,E2 -13794.904} C_VEL
LIN {X 0,Y 360.738,Z 377.904,A -85,B 0,C 180,E1 -13796.061,E2 -13796.061} C_VEL
LIN {X 0,Y 362.268,Z 363.295,A -85,B 0,C 180,E1 -13796.99,E2 -13796.99} C_VEL
LIN {X 0,Y 363.563,Z 348.657,A -85,B 0,C 180,E1 -13797.681,E2 -13797.681} C_VEL
LIN {X 0,Y 364.521,Z 332.92,A -85,B 0,C 180,E1 -13798.188,E2 -13798.188} C_VEL
LIN {X 0,Y 367.672,Z 218.609,A -85,B 0,C 180,E1 -13800.456,E2 -13800.456} C_VEL
LIN {X 0,Y 367.716,Z 210.147,A -85,B 0,C 180,E1 -13800.639,E2 -13800.639} C_VEL
LIN {X 0,Y 365.04,Z 196.57,A -85,B 0,C 180,E1 -13801.193,E2 -13801.193} C_VEL
LIN {X 0,Y 357.409,Z 179.524,A -85,B 0,C 180,E1 -13802.33,E2 -13802.33} C_VEL
LIN {X 0,Y 351.924,Z 168.071,A -85,B 0,C 180,E1 -13803.211,E2 -13803.211} C_VEL
LIN {X 0,Y 349.046,Z 157.298,A -85,B 0,C 180,E1 -13806.017,E2 -13806.017} C_VEL
LIN {X 0,Y 347.81,Z 152.83,A -85,B 0,C 180,E1 -13807.315,E2 -13807.315} C_VEL
LIN {X 0,Y 347.732,Z 152.781,A -85,B 0,C 180,E1 -13810.297,E2 -13810.297} C_VEL
LIN {X 0,Y 347.723,Z 152.773,A -85,B 0,C 180,E1 -13813.408,E2 -13813.408} C_VEL
LIN {X 0,Y 347.725,Z 152.796,A -85,B 0,C 180,E1 -13816.686,E2 -13816.686} C_VEL
LIN {X 0,Y 347.747,Z 152.762,A -85,B 0,C 180,E1 -13820.173,E2 -13820.173} C_VEL
LIN {X 0,Y 347.762,Z 152.791,A -85,B 0,C 180,E1 -13822.679,E2 -13822.679} C_VEL
LIN {X 0,Y 347.748,Z 152.748,A -85,B 0,C 180,E1 -13825.956,E2 -13825.956} C_VEL
LIN {X 0,Y 347.764,Z 152.775,A -85,B 0,C 180,E1 -13829.654,E2 -13829.654} C_VEL
LIN {X 0,Y 347.852,Z 152.773,A -85,B 0,C 180,E1 -13832.745,E2 -13832.745} C_VEL
LIN {X 0,Y 347.79,Z 152.786,A -85,B 0,C 180,E1 -13836.162,E2 -13836.162} C_VEL
LIN {X 0,Y 347.813,Z 152.775,A -85,B 0,C 180,E1 -13839.91,E2 -13839.91} C_VEL
LIN {X 0,Y 347.867,Z 152.777,A -85,B 0,C 180,E1 -13842.359,E2 -13842.359} C_VEL
LIN {X 0,Y 347.899,Z 152.768,A -85,B 0,C 180,E1 -13845.971,E2 -13845.971} C_VEL
LIN {X 0,Y 347.898,Z 152.76,A -85,B 0,C 180,E1 -13849.525,E2 -13849.525} C_VEL
LIN {X 0,Y 348.065,Z 152.753,A -85,B 0,C 180,E1 -13853.042,E2 -13853.042} C_VEL
LIN {X 0,Y 348.204,Z 152.725,A -85,B 0,C 180,E1 -13857.687,E2 -13857.687} C_VEL
LIN {X 0,Y 348.304,Z 152.721,A -85,B 0,C 180,E1 -13860,E2 -13860} C_VEL
LIN {X 0,Y 348.195,Z 152.717,A -85,B 0,C 180,E1 -13862.314,E2 -13862.314} C_VEL
LIN {X 0,Y 348.068,Z 152.745,A -85,B 0,C 180,E1 -13866.959,E2 -13866.959} C_VEL
LIN {X 0,Y 347.898,Z 152.771,A -85,B 0,C 180,E1 -13870.475,E2 -13870.475} C_VEL
LIN {X 0,Y 347.9,Z 152.757,A -85,B 0,C 180,E1 -13874.15,E2 -13874.15} C_VEL
LIN {X 0,Y 347.83,Z 152.777,A -85,B 0,C 180,E1 -13878.259,E2 -13878.259} C_VEL
LIN {X 0,Y 347.768,Z 152.784,A -85,B 0,C 180,E1 -13881.626,E2 -13881.626} C_VEL
LIN {X 0,Y 347.739,Z 152.779,A -85,B 0,C 180,E1 -13885.114,E2 -13885.114} C_VEL
LIN {X 0,Y 347.736,Z 152.797,A -85,B 0,C 180,E1 -13887.7,E2 -13887.7} C_VEL
LIN {X 0,Y 347.736,Z 152.763,A -85,B 0,C 180,E1 -13890.349,E2 -13890.349} C_VEL
LIN {X 0,Y 347.749,Z 152.76,A -85,B 0,C 180,E1 -13894.044,E2 -13894.044} C_VEL
LIN {X 0,Y 347.757,Z 152.788,A -85,B 0,C 180,E1 -13897.322,E2 -13897.322} C_VEL
LIN {X 0,Y 347.741,Z 152.766,A -85,B 0,C 180,E1 -13901.601,E2 -13901.601} C_VEL
LIN {X 0,Y 347.702,Z 152.783,A -85,B 0,C 180,E1 -13905.028,E2 -13905.028} C_VEL
LIN {X 0,Y 347.74,Z 152.796,A -85,B 0,C 180,E1 -13908.399,E2 -13908.399} C_VEL
LIN {X 0,Y 347.756,Z 152.786,A -85,B 0,C 180,E1 -13912.678,E2 -13912.678} C_VEL
LIN {X 0,Y 347.792,Z 152.91,A -85,B 0,C 180,E1 -13913.93,E2 -13913.93} C_VEL
LIN {X 0,Y 350.309,Z 162.088,A -85,B 0,C 180,E1 -13916.54,E2 -13916.54} C_VEL
LIN {X 0,Y 350.698,Z 163.329,A -85,B 0,C 180,E1 -13916.752,E2 -13916.752} C_VEL
LIN {X 0,Y 359.632,Z 181.428,A -85,B 0,C 180,E1 -13918.114,E2 -13918.114} C_VEL
LIN {X 0,Y 367.482,Z 199.445,A -85,B 0,C 180,E1 -13919.277,E2 -13919.277} C_VEL
LIN {X 0,Y 368.05,Z 203.815,A -85,B 0,C 180,E1 -13919.427,E2 -13919.427} C_VEL
LIN {X 0,Y 364.664,Z 326.686,A -85,B 0,C 180,E1 -13921.863,E2 -13921.863} C_VEL
LIN {X 0,Y 363.813,Z 341.581,A -85,B 0,C 180,E1 -13922.34,E2 -13922.34} C_VEL
LIN {X 0,Y 362.722,Z 354.961,A -85,B 0,C 180,E1 -13922.954,E2 -13922.954} C_VEL
LIN {X 0,Y 361.197,Z 370.076,A -85,B 0,C 180,E1 -13923.882,E2 -13923.882} C_VEL
LIN {X 0,Y 359.435,Z 384.079,A -85,B 0,C 180,E1 -13924.987,E2 -13924.987} C_VEL
LIN {X 0,Y 357.624,Z 396.881,A -85,B 0,C 180,E1 -13926.243,E2 -13926.243} C_VEL
LIN {X 0,Y 355.495,Z 409.781,A -85,B 0,C 180,E1 -13927.784,E2 -13927.784} C_VEL
LIN {X 0,Y 353.81,Z 420.564,A -85,B 0,C 180,E1 -13929.355,E2 -13929.355} C_VEL
LIN {X 0,Y 352.045,Z 430.535,A -85,B 0,C 180,E1 -13931.07,E2 -13931.07} C_VEL
LIN {X 0,Y 350.385,Z 440.275,A -85,B 0,C 180,E1 -13933.092,E2 -13933.092} C_VEL
LIN {X 0,Y 348.906,Z 448.702,A -85,B 0,C 180,E1 -13935.209,E2 -13935.209} C_VEL
LIN {X 0,Y 348.058,Z 455.092,A -85,B 0,C 180,E1 -13937.167,E2 -13937.167} C_VEL
LIN {X 0,Y 347.131,Z 461.298,A -85,B 0,C 180,E1 -13939.501,E2 -13939.501} C_VEL
LIN {X 0,Y 346.562,Z 466.09,A -85,B 0,C 180,E1 -13941.839,E2 -13941.839} C_VEL
LIN {X 0,Y 346.289,Z 469.602,A -85,B 0,C 180,E1 -13944.176,E2 -13944.176} C_VEL
LIN {X 0,Y 346.142,Z 471.924,A -85,B 0,C 180,E1 -13946.508,E2 -13946.508} C_VEL
LIN {X 0,Y 346.058,Z 473.11,A -85,B 0,C 180,E1 -13948.836,E2 -13948.836} C_VEL
LIN {X 0,Y 346.059,Z 473.125,A -85,B 0,C 180,E1 -13951.164,E2 -13951.164} C_VEL
LIN {X 0,Y 346.14,Z 471.999,A -85,B 0,C 180,E1 -13953.492,E2 -13953.492} C_VEL
LIN {X 0,Y 346.25,Z 469.557,A -85,B 0,C 180,E1 -13955.969,E2 -13955.969} C_VEL
LIN {X 0,Y 346.685,Z 465.216,A -85,B 0,C 180,E1 -13958.745,E2 -13958.745} C_VEL
LIN {X 0,Y 347.265,Z 460.128,A -85,B 0,C 180,E1 -13961.085,E2 -13961.085} C_VEL
LIN {X 0,Y 348.262,Z 453.612,A -85,B 0,C 180,E1 -13963.419,E2 -13963.419} C_VEL
LIN {X 0,Y 349.473,Z 445.471,A -85,B 0,C 180,E1 -13965.753,E2 -13965.753} C_VEL
LIN {X 0,Y 350.984,Z 436.778,A -85,B 0,C 180,E1 -13967.78,E2 -13967.78} C_VEL
LIN {X 0,Y 352.533,Z 427.947,A -85,B 0,C 180,E1 -13969.507,E2 -13969.507} C_VEL
LIN {X 0,Y 354.147,Z 418.14,A -85,B 0,C 180,E1 -13971.139,E2 -13971.139} C_VEL
LIN {X 0,Y 356.191,Z 406.205,A -85,B 0,C 180,E1 -13972.782,E2 -13972.782} C_VEL
LIN {X 0,Y 357.359,Z 398.766,A -85,B 0,C 180,E1 -13973.657,E2 -13973.657} C_VEL
LIN {X 0,Y 357.441,Z 394.012,A -85,B 0,C 180,E1 -13974.22,E2 -13974.22} C_VEL
LIN {X 0,Y 354.634,Z 379.849,A -85,B 0,C 180,E1 -13975.916,E2 -13975.916} C_VEL
LIN {X 0,Y 354.38,Z 374.75,A -85,B 0,C 180,E1 -13976.392,E2 -13976.392} C_VEL
LIN {X 0,Y 354.533,Z 372.979,A -85,B 0,C 180,E1 -13976.528,E2 -13976.528} C_VEL
LIN {X 0,Y 356.139,Z 358.454,A -85,B 0,C 180,E1 -13977.487,E2 -13977.487} C_VEL
LIN {X 0,Y 357.443,Z 343.221,A -85,B 0,C 180,E1 -13978.237,E2 -13978.237} C_VEL
LIN {X 0,Y 358.413,Z 327.851,A -85,B 0,C 180,E1 -13978.753,E2 -13978.753} C_VEL
LIN {X 0,Y 361.507,Z 222.915,A -85,B 0,C 180,E1 -13980.866,E2 -13980.866} C_VEL
LIN {X 0,Y 361.861,Z 202.813,A -85,B 0,C 180,E1 -13981.289,E2 -13981.289} C_VEL
LIN {X 0,Y 354.974,Z 186.635,A -85,B 0,C 180,E1 -13982.347,E2 -13982.347} C_VEL
LIN {X 0,Y 346.616,Z 169.524,A -85,B 0,C 180,E1 -13983.644,E2 -13983.644} C_VEL
LIN {X 0,Y 343.231,Z 162.779,A -85,B 0,C 180,E1 -13984.237,E2 -13984.237} C_VEL
LIN {X 0,Y 340.73,Z 153.822,A -85,B 0,C 180,E1 -13986.831,E2 -13986.831} C_VEL
LIN {X 0,Y 340.651,Z 153.661,A -85,B 0,C 180,E1 -13990.239,E2 -13990.239} C_VEL
LIN {X 0,Y 340.672,Z 153.662,A -85,B 0,C 180,E1 -13992.905,E2 -13992.905} C_VEL
LIN {X 0,Y 340.672,Z 153.673,A -85,B 0,C 180,E1 -13997.095,E2 -13997.095} C_VEL
LIN {X 0,Y 340.655,Z 153.634,A -85,B 0,C 180,E1 -14000.241,E2 -14000.241} C_VEL
LIN {X 0,Y 340.71,Z 153.67,A -85,B 0,C 180,E1 -14003.56,E2 -14003.56} C_VEL
LIN {X 0,Y 340.693,Z 153.637,A -85,B 0,C 180,E1 -14006.153,E2 -14006.153} C_VEL
LIN {X 0,Y 340.72,Z 153.642,A -85,B 0,C 180,E1 -14010.035,E2 -14010.035} C_VEL
LIN {X 0,Y 340.719,Z 153.666,A -85,B 0,C 180,E1 -14013.013,E2 -14013.013} C_VEL
LIN {X 0,Y 340.707,Z 153.669,A -85,B 0,C 180,E1 -14016.925,E2 -14016.925} C_VEL
LIN {X 0,Y 340.736,Z 153.653,A -85,B 0,C 180,E1 -14020.73,E2 -14020.73} C_VEL
LIN {X 0,Y 340.8,Z 153.647,A -85,B 0,C 180,E1 -14024.449,E2 -14024.449} C_VEL
LIN {X 0,Y 340.844,Z 153.645,A -85,B 0,C 180,E1 -14026.89,E2 -14026.89} C_VEL
LIN {X 0,Y 340.884,Z 153.635,A -85,B 0,C 180,E1 -14030.506,E2 -14030.506} C_VEL
LIN {X 0,Y 341.028,Z 153.631,A -85,B 0,C 180,E1 -14034.086,E2 -14034.086} C_VEL
LIN {X 0,Y 341.131,Z 153.596,A -85,B 0,C 180,E1 -14037.638,E2 -14037.638} C_VEL
LIN {X 0,Y 341.237,Z 153.602,A -85,B 0,C 180,E1 -14040,E2 -14040} C_VEL
LIN {X 0,Y 341.159,Z 153.602,A -85,B 0,C 180,E1 -14042.361,E2 -14042.361} C_VEL
LIN {X 0,Y 341.011,Z 153.633,A -85,B 0,C 180,E1 -14047.103,E2 -14047.103} C_VEL
LIN {X 0,Y 340.85,Z 153.639,A -85,B 0,C 180,E1 -14050.694,E2 -14050.694} C_VEL
LIN {X 0,Y 340.865,Z 153.642,A -85,B 0,C 180,E1 -14054.325,E2 -14054.325} C_VEL
LIN {X 0,Y 340.838,Z 153.654,A -85,B 0,C 180,E1 -14058.466,E2 -14058.466} C_VEL
LIN {X 0,Y 340.719,Z 153.657,A -85,B 0,C 180,E1 -14061.841,E2 -14061.841} C_VEL
LIN {X 0,Y 340.773,Z 153.647,A -85,B 0,C 180,E1 -14065.664,E2 -14065.664} C_VEL
LIN {X 0,Y 340.742,Z 153.666,A -85,B 0,C 180,E1 -14068.319,E2 -14068.319} C_VEL
LIN {X 0,Y 340.704,Z 153.64,A -85,B 0,C 180,E1 -14071.044,E2 -14071.044} C_VEL
LIN {X 0,Y 340.718,Z 153.648,A -85,B 0,C 180,E1 -14075.279,E2 -14075.279} C_VEL
LIN {X 0,Y 340.71,Z 153.657,A -85,B 0,C 180,E1 -14078.386,E2 -14078.386} C_VEL
LIN {X 0,Y 340.699,Z 153.653,A -85,B 0,C 180,E1 -14082.045,E2 -14082.045} C_VEL
LIN {X 0,Y 340.652,Z 153.651,A -85,B 0,C 180,E1 -14086.227,E2 -14086.227} C_VEL
LIN {X 0,Y 340.688,Z 153.657,A -85,B 0,C 180,E1 -14089.753,E2 -14089.753} C_VEL
LIN {X 0,Y 340.768,Z 153.823,A -85,B 0,C 180,E1 -14092.065,E2 -14092.065} C_VEL
LIN {X 0,Y 344.243,Z 166.312,A -85,B 0,C 180,E1 -14095.566,E2 -14095.566} C_VEL
LIN {X 0,Y 344.826,Z 168.364,A -85,B 0,C 180,E1 -14096.022,E2 -14096.022} C_VEL
LIN {X 0,Y 354.231,Z 187.868,A -85,B 0,C 180,E1 -14097.52,E2 -14097.52} C_VEL
LIN {X 0,Y 359.597,Z 200.364,A -85,B 0,C 180,E1 -14098.349,E2 -14098.349} C_VEL
LIN {X 0,Y 361.811,Z 212.203,A -85,B 0,C 180,E1 -14098.834,E2 -14098.834} C_VEL
LIN {X 0,Y 358.377,Z 332.043,A -85,B 0,C 180,E1 -14101.244,E2 -14101.244} C_VEL
LIN {X 0,Y 357.44,Z 347.163,A -85,B 0,C 180,E1 -14101.723,E2 -14101.723} C_VEL
LIN {X 0,Y 356.005,Z 362.614,A -85,B 0,C 180,E1 -14102.44,E2 -14102.44} C_VEL
LIN {X 0,Y 354.537,Z 376.796,A -85,B 0,C 180,E1 -14103.346,E2 -14103.346} C_VEL
LIN {X 0,Y 352.903,Z 389.158,A -85,B 0,C 180,E1 -14104.332,E2 -14104.332} C_VEL
LIN {X 0,Y 350.875,Z 402.149,A -85,B 0,C 180,E1 -14105.599,E2 -14105.599} C_VEL
LIN {X 0,Y 348.692,Z 415.216,A -85,B 0,C 180,E1 -14107.17,E2 -14107.17} C_VEL
LIN {X 0,Y 346.789,Z 426.286,A -85,B 0,C 180,E1 -14108.785,E2 -14108.785} C_VEL
LIN {X 0,Y 344.904,Z 436.989,A -85,B 0,C 180,E1 -14110.663,E2 -14110.663} C_VEL
LIN {X 0,Y 343.135,Z 446.72,A -85,B 0,C 180,E1 -14112.723,E2 -14112.723} C_VEL
LIN {X 0,Y 341.938,Z 453.761,A -85,B 0,C 180,E1 -14114.503,E2 -14114.503} C_VEL
LIN {X 0,Y 340.762,Z 461.552,A -85,B 0,C 180,E1 -14116.887,E2 -14116.887} C_VEL
LIN {X 0,Y 339.838,Z 467.748,A -85,B 0,C 180,E1 -14119.273,E2 -14119.273} C_VEL
LIN {X 0,Y 339.392,Z 472.541,A -85,B 0,C 180,E1 -14121.665,E2 -14121.665} C_VEL
LIN {X 0,Y 339.125,Z 476.14,A -85,B 0,C 180,E1 -14124.125,E2 -14124.125} C_VEL
LIN {X 0,Y 339.03,Z 478.36,A -85,B 0,C 180,E1 -14126.434,E2 -14126.434} C_VEL
LIN {X 0,Y 338.952,Z 479.52,A -85,B 0,C 180,E1 -14128.812,E2 -14128.812} C_VEL
LIN {X 0,Y 338.952,Z 479.517,A -85,B 0,C 180,E1 -14131.188,E2 -14131.188} C_VEL
LIN {X 0,Y 339.03,Z 478.346,A -85,B 0,C 180,E1 -14133.565,E2 -14133.565} C_VEL
LIN {X 0,Y 339.128,Z 476.029,A -85,B 0,C 180,E1 -14135.948,E2 -14135.948} C_VEL
LIN {X 0,Y 339.393,Z 472.516,A -85,B 0,C 180,E1 -14138.335,E2 -14138.335} C_VEL
LIN {X 0,Y 339.833,Z 467.716,A -85,B 0,C 180,E1 -14140.727,E2 -14140.727} C_VEL
LIN {X 0,Y 340.751,Z 461.501,A -85,B 0,C 180,E1 -14143.113,E2 -14143.113} C_VEL
LIN {X 0,Y 341.926,Z 453.695,A -85,B 0,C 180,E1 -14145.498,E2 -14145.498} C_VEL
LIN {X 0,Y 343.373,Z 445.393,A -85,B 0,C 180,E1 -14147.572,E2 -14147.572} C_VEL
LIN {X 0,Y 345.236,Z 435.39,A -85,B 0,C 180,E1 -14149.627,E2 -14149.627} C_VEL
LIN {X 0,Y 346.948,Z 425.156,A -85,B 0,C 180,E1 -14151.384,E2 -14151.384} C_VEL
LIN {X 0,Y 349.104,Z 412.96,A -85,B 0,C 180,E1 -14153.114,E2 -14153.114} C_VEL
LIN {X 0,Y 351.062,Z 400.715,A -85,B 0,C 180,E1 -14154.544,E2 -14154.544} C_VEL
LIN {X 0,Y 353.107,Z 387.385,A -85,B 0,C 180,E1 -14155.81,E2 -14155.81} C_VEL
LIN {X 0,Y 354.98,Z 372.52,A -85,B 0,C 180,E1 -14156.941,E2 -14156.941} C_VEL
LIN {X 0,Y 356.464,Z 357.759,A -85,B 0,C 180,E1 -14157.801,E2 -14157.801} C_VEL
LIN {X 0,Y 357.758,Z 342.162,A -85,B 0,C 180,E1 -14158.449,E2 -14158.449} C_VEL
LIN {X 0,Y 358.541,Z 326.811,A -85,B 0,C 180,E1 -14158.861,E2 -14158.861} C_VEL
LIN {X 0,Y 361.716,Z 213.141,A -85,B 0,C 180,E1 -14161.134,E2 -14161.134} C_VEL
LIN {X 0,Y 360.742,Z 206.553,A -85,B 0,C 180,E1 -14161.377,E2 -14161.377} C_VEL
LIN {X 0,Y 359.219,Z 199.287,A -85,B 0,C 180,E1 -14161.692,E2 -14161.692} C_VEL
LIN {X 0,Y 350.998,Z 181.008,A -85,B 0,C 180,E1 -14162.957,E2 -14162.957} C_VEL
LIN {X 0,Y 344.688,Z 167.988,A -85,B 0,C 180,E1 -14164.002,E2 -14164.002} C_VEL
LIN {X 0,Y 341.221,Z 155.454,A -85,B 0,C 180,E1 -14167.415,E2 -14167.415} C_VEL
LIN {X 0,Y 340.746,Z 153.7,A -85,B 0,C 180,E1 -14167.991,E2 -14167.991} C_VEL
LIN {X 0,Y 340.699,Z 153.667,A -85,B 0,C 180,E1 -14172.046,E2 -14172.046} C_VEL
LIN {X 0,Y 340.652,Z 153.679,A -85,B 0,C 180,E1 -14176.227,E2 -14176.227} C_VEL
LIN {X 0,Y 340.687,Z 153.638,A -85,B 0,C 180,E1 -14179.753,E2 -14179.753} C_VEL
LIN {X 0,Y 340.705,Z 153.672,A -85,B 0,C 180,E1 -14183.259,E2 -14183.259} C_VEL
LIN {X 0,Y 340.692,Z 153.623,A -85,B 0,C 180,E1 -14186.153,E2 -14186.153} C_VEL
LIN {X 0,Y 340.775,Z 153.658,A -85,B 0,C 180,E1 -14190.333,E2 -14190.333} C_VEL
LIN {X 0,Y 340.805,Z 153.647,A -85,B 0,C 180,E1 -14193.02,E2 -14193.02} C_VEL
LIN {X 0,Y 340.73,Z 153.667,A -85,B 0,C 180,E1 -14196.927,E2 -14196.927} C_VEL
LIN {X 0,Y 340.791,Z 153.655,A -85,B 0,C 180,E1 -14200.734,E2 -14200.734} C_VEL
LIN {X 0,Y 340.787,Z 153.649,A -85,B 0,C 180,E1 -14203.219,E2 -14203.219} C_VEL
LIN {X 0,Y 340.845,Z 153.653,A -85,B 0,C 180,E1 -14206.891,E2 -14206.891} C_VEL
LIN {X 0,Y 340.883,Z 153.628,A -85,B 0,C 180,E1 -14210.507,E2 -14210.507} C_VEL
LIN {X 0,Y 341.026,Z 153.628,A -85,B 0,C 180,E1 -14214.086,E2 -14214.086} C_VEL
LIN {X 0,Y 341.165,Z 153.601,A -85,B 0,C 180,E1 -14217.639,E2 -14217.639} C_VEL
LIN {X 0,Y 341.256,Z 153.599,A -85,B 0,C 180,E1 -14220,E2 -14220} C_VEL
LIN {X 0,Y 341.133,Z 153.596,A -85,B 0,C 180,E1 -14222.362,E2 -14222.362} C_VEL
LIN {X 0,Y 341.002,Z 153.627,A -85,B 0,C 180,E1 -14226.5,E2 -14226.5} C_VEL
LIN {X 0,Y 340.883,Z 153.635,A -85,B 0,C 180,E1 -14229.494,E2 -14229.494} C_VEL
LIN {X 0,Y 340.846,Z 153.646,A -85,B 0,C 180,E1 -14233.11,E2 -14233.11} C_VEL
LIN {X 0,Y 340.775,Z 153.66,A -85,B 0,C 180,E1 -14236.782,E2 -14236.782} C_VEL
LIN {X 0,Y 340.736,Z 153.653,A -85,B 0,C 180,E1 -14239.27,E2 -14239.27} C_VEL
LIN {X 0,Y 340.706,Z 153.669,A -85,B 0,C 180,E1 -14243.075,E2 -14243.075} C_VEL
LIN {X 0,Y 340.718,Z 153.666,A -85,B 0,C 180,E1 -14246.988,E2 -14246.988} C_VEL
LIN {X 0,Y 340.691,Z 153.625,A -85,B 0,C 180,E1 -14251.046,E2 -14251.046} C_VEL
LIN {X 0,Y 340.718,Z 153.661,A -85,B 0,C 180,E1 -14255.279,E2 -14255.279} C_VEL
LIN {X 0,Y 340.694,Z 153.648,A -85,B 0,C 180,E1 -14258.382,E2 -14258.382} C_VEL
LIN {X 0,Y 340.694,Z 153.651,A -85,B 0,C 180,E1 -14262.044,E2 -14262.044} C_VEL
LIN {X 0,Y 340.65,Z 153.655,A -85,B 0,C 180,E1 -14266.227,E2 -14266.227} C_VEL
LIN {X 0,Y 340.67,Z 153.672,A -85,B 0,C 180,E1 -14268.688,E2 -14268.688} C_VEL
LIN {X 0,Y 340.73,Z 153.658,A -85,B 0,C 180,E1 -14272.892,E2 -14272.892} C_VEL
LIN {X 0,Y 340.775,Z 153.977,A -85,B 0,C 180,E1 -14273.366,E2 -14273.366} C_VEL
LIN {X 0,Y 343.336,Z 162.971,A -85,B 0,C 180,E1 -14275.914,E2 -14275.914} C_VEL
LIN {X 0,Y 353.09,Z 182.612,A -85,B 0,C 180,E1 -14277.477,E2 -14277.477} C_VEL
LIN {X 0,Y 360.281,Z 198.84,A -85,B 0,C 180,E1 -14278.578,E2 -14278.578} C_VEL
LIN {X 0,Y 361.761,Z 202.77,A -85,B 0,C 180,E1 -14278.811,E2 -14278.811} C_VEL
LIN {X 0,Y 361.797,Z 209.617,A -85,B 0,C 180,E1 -14278.97,E2 -14278.97} C_VEL
LIN {X 0,Y 358.441,Z 326.773,A -85,B 0,C 180,E1 -14281.33,E2 -14281.33} C_VEL
LIN {X 0,Y 357.545,Z 341.66,A -85,B 0,C 180,E1 -14281.812,E2 -14281.812} C_VEL
LIN {X 0,Y 356.35,Z 355.69,A -85,B 0,C 180,E1 -14282.469,E2 -14282.469} C_VEL
LIN {X 0,Y 354.816,Z 370.15,A -85,B 0,C 180,E1 -14283.375,E2 -14283.375} C_VEL
LIN {X 0,Y 353.005,Z 384.151,A -85,B 0,C 180,E1 -14284.499,E2 -14284.499} C_VEL
LIN {X 0,Y 351.105,Z 396.952,A -85,B 0,C 180,E1 -14285.774,E2 -14285.774} C_VEL
LIN {X 0,Y 348.909,Z 409.851,A -85,B 0,C 180,E1 -14287.342,E2 -14287.342} C_VEL
LIN {X 0,Y 347.144,Z 420.633,A -85,B 0,C 180,E1 -14288.94,E2 -14288.94} C_VEL
LIN {X 0,Y 345.277,Z 430.605,A -85,B 0,C 180,E1 -14290.685,E2 -14290.685} C_VEL
LIN {X 0,Y 343.538,Z 440.344,A -85,B 0,C 180,E1 -14292.744,E2 -14292.744} C_VEL
LIN {X 0,Y 342.275,Z 447.369,A -85,B 0,C 180,E1 -14294.518,E2 -14294.518} C_VEL
LIN {X 0,Y 341.097,Z 455.161,A -85,B 0,C 180,E1 -14296.9,E2 -14296.9} C_VEL
LIN {X 0,Y 340.107,Z 461.366,A -85,B 0,C 180,E1 -14299.282,E2 -14299.282} C_VEL
LIN {X 0,Y 339.52,Z 466.158,A -85,B 0,C 180,E1 -14301.669,E2 -14301.669} C_VEL
LIN {X 0,Y 339.21,Z 469.669,A -85,B 0,C 180,E1 -14304.054,E2 -14304.054} C_VEL
LIN {X 0,Y 339.069,Z 471.991,A -85,B 0,C 180,E1 -14306.435,E2 -14306.435} C_VEL
LIN {X 0,Y 338.964,Z 473.177,A -85,B 0,C 180,E1 -14308.812,E2 -14308.812} C_VEL
LIN {X 0,Y 338.965,Z 473.191,A -85,B 0,C 180,E1 -14311.188,E2 -14311.188} C_VEL
LIN {X 0,Y 339.067,Z 472.065,A -85,B 0,C 180,E1 -14313.565,E2 -14313.565} C_VEL
LIN {X 0,Y 339.17,Z 469.801,A -85,B 0,C 180,E1 -14315.947,E2 -14315.947} C_VEL
LIN {X 0,Y 339.513,Z 466.343,A -85,B 0,C 180,E1 -14318.332,E2 -14318.332} C_VEL
LIN {X 0,Y 340.074,Z 461.611,A -85,B 0,C 180,E1 -14320.719,E2 -14320.719} C_VEL
LIN {X 0,Y 341.043,Z 455.48,A -85,B 0,C 180,E1 -14323.102,E2 -14323.102} C_VEL
LIN {X 0,Y 342.21,Z 447.763,A -85,B 0,C 180,E1 -14325.485,E2 -14325.485} C_VEL
LIN {X 0,Y 343.698,Z 439.536,A -85,B 0,C 180,E1 -14327.554,E2 -14327.554} C_VEL
LIN {X 0,Y 345.5,Z 429.627,A -85,B 0,C 180,E1 -14329.611,E2 -14329.611} C_VEL
LIN {X 0,Y 347.026,Z 421.318,A -85,B 0,C 180,E1 -14331.056,E2 -14331.056} C_VEL
LIN {X 0,Y 349.066,Z 409.512,A -85,B 0,C 180,E1 -14332.804,E2 -14332.804} C_VEL
LIN {X 0,Y 351.181,Z 396.542,A -85,B 0,C 180,E1 -14334.378,E2 -14334.378} C_VEL
LIN {X 0,Y 353.11,Z 383.66,A -85,B 0,C 180,E1 -14335.651,E2 -14335.651} C_VEL
LIN {X 0,Y 354.533,Z 372.979,A -85,B 0,C 180,E1 -14336.528,E2 -14336.528} C_VEL
LIN {X 0,Y 354.687,Z 367.672,A -85,B 0,C 180,E1 -14336.946,E2 -14336.946} C_VEL
LIN {X 0,Y 353.161,Z 359.07,A -85,B 0,C 180,E1 -14337.698,E2 -14337.698} C_VEL
LIN {X 0,Y 351.383,Z 350.317,A -85,B 0,C 180,E1 -14338.395,E2 -14338.395} C_VEL
LIN {X 0,Y 351.104,Z 344.769,A -85,B 0,C 180,E1 -14338.717,E2 -14338.717} C_VEL
LIN {X 0,Y 352.165,Z 329.122,A -85,B 0,C 180,E1 -14339.271,E2 -14339.271} C_VEL
LIN {X 0,Y 353.938,Z 274.252,A -85,B 0,C 180,E1 -14340.411,E2 -14340.411} C_VEL
LIN {X 0,Y 355.861,Z 204.759,A -85,B 0,C 180,E1 -14341.833,E2 -14341.833} C_VEL
LIN {X 0,Y 348.17,Z 187.183,A -85,B 0,C 180,E1 -14343.046,E2 -14343.046} C_VEL
LIN {X 0,Y 339.313,Z 169.313,A -85,B 0,C 180,E1 -14344.475,E2 -14344.475} C_VEL
LIN {X 0,Y 336.062,Z 162.991,A -85,B 0,C 180,E1 -14345.055,E2 -14345.055} C_VEL
LIN {X 0,Y 333.698,Z 154.714,A -85,B 0,C 180,E1 -14347.52,E2 -14347.52} C_VEL
LIN {X 0,Y 333.603,Z 154.542,A -85,B 0,C 180,E1 -14350.774,E2 -14350.774} C_VEL
LIN {X 0,Y 333.59,Z 154.533,A -85,B 0,C 180,E1 -14354.25,E2 -14354.25} C_VEL
LIN {X 0,Y 333.636,Z 154.541,A -85,B 0,C 180,E1 -14357.617,E2 -14357.617} C_VEL
LIN {X 0,Y 333.617,Z 154.518,A -85,B 0,C 180,E1 -14361.21,E2 -14361.21} C_VEL
LIN {X 0,Y 333.676,Z 154.547,A -85,B 0,C 180,E1 -14363.861,E2 -14363.861} C_VEL
LIN {X 0,Y 333.644,Z 154.495,A -85,B 0,C 180,E1 -14367.413,E2 -14367.413} C_VEL
LIN {X 0,Y 333.653,Z 154.538,A -85,B 0,C 180,E1 -14371.022,E2 -14371.022} C_VEL
LIN {X 0,Y 333.665,Z 154.531,A -85,B 0,C 180,E1 -14375.086,E2 -14375.086} C_VEL
LIN {X 0,Y 333.665,Z 154.537,A -85,B 0,C 180,E1 -14379.018,E2 -14379.018} C_VEL
LIN {X 0,Y 333.742,Z 154.53,A -85,B 0,C 180,E1 -14381.586,E2 -14381.586} C_VEL
LIN {X 0,Y 333.808,Z 154.511,A -85,B 0,C 180,E1 -14385.578,E2 -14385.578} C_VEL
LIN {X 0,Y 333.82,Z 154.527,A -85,B 0,C 180,E1 -14389.077,E2 -14389.077} C_VEL
LIN {X 0,Y 333.966,Z 154.499,A -85,B 0,C 180,E1 -14392.746,E2 -14392.746} C_VEL
LIN {X 0,Y 333.793,Z 154.531,A -85,B 0,C 180,E1 -14395.169,E2 -14395.169} C_VEL
LIN {X 0,Y 334.072,Z 154.475,A -85,B 0,C 180,E1 -14397.588,E2 -14397.588} C_VEL
LIN {X 0,Y 334.189,Z 154.48,A -85,B 0,C 180,E1 -14400,E2 -14400} C_VEL
LIN {X 0,Y 334.096,Z 154.481,A -85,B 0,C 180,E1 -14402.411,E2 -14402.411} C_VEL
LIN {X 0,Y 333.999,Z 154.503,A -85,B 0,C 180,E1 -14406.039,E2 -14406.039} C_VEL
LIN {X 0,Y 333.822,Z 154.507,A -85,B 0,C 180,E1 -14409.696,E2 -14409.696} C_VEL
LIN {X 0,Y 333.799,Z 154.528,A -85,B 0,C 180,E1 -14413.391,E2 -14413.391} C_VEL
LIN {X 0,Y 333.748,Z 154.53,A -85,B 0,C 180,E1 -14417.146,E2 -14417.146} C_VEL
LIN {X 0,Y 333.733,Z 154.531,A -85,B 0,C 180,E1 -14419.69,E2 -14419.69} C_VEL
LIN {X 0,Y 333.67,Z 154.546,A -85,B 0,C 180,E1 -14423.59,E2 -14423.59} C_VEL
LIN {X 0,Y 333.736,Z 154.522,A -85,B 0,C 180,E1 -14426.246,E2 -14426.246} C_VEL
LIN {X 0,Y 333.712,Z 154.54,A -85,B 0,C 180,E1 -14428.972,E2 -14428.972} C_VEL
LIN {X 0,Y 333.644,Z 154.496,A -85,B 0,C 180,E1 -14432.587,E2 -14432.587} C_VEL
LIN {X 0,Y 333.676,Z 154.541,A -85,B 0,C 180,E1 -14436.139,E2 -14436.139} C_VEL
LIN {X 0,Y 333.647,Z 154.522,A -85,B 0,C 180,E1 -14439.192,E2 -14439.192} C_VEL
LIN {X 0,Y 333.633,Z 154.542,A -85,B 0,C 180,E1 -14442.5,E2 -14442.5} C_VEL
LIN {X 0,Y 333.596,Z 154.529,A -85,B 0,C 180,E1 -14445.955,E2 -14445.955} C_VEL
LIN {X 0,Y 333.647,Z 154.538,A -85,B 0,C 180,E1 -14449.315,E2 -14449.315} C_VEL
LIN {X 0,Y 333.696,Z 154.72,A -85,B 0,C 180,E1 -14451.368,E2 -14451.368} C_VEL
LIN {X 0,Y 336.718,Z 165.446,A -85,B 0,C 180,E1 -14454.49,E2 -14454.49} C_VEL
LIN {X 0,Y 337.545,Z 168.189,A -85,B 0,C 180,E1 -14455.178,E2 -14455.178} C_VEL
LIN {X 0,Y 346.204,Z 185.69,A -85,B 0,C 180,E1 -14456.618,E2 -14456.618} C_VEL
LIN {X 0,Y 353.791,Z 202.839,A -85,B 0,C 180,E1 -14457.827,E2 -14457.827} C_VEL
LIN {X 0,Y 355.736,Z 214.137,A -85,B 0,C 180,E1 -14458.286,E2 -14458.286} C_VEL
LIN {X 0,Y 352.131,Z 333.497,A -85,B 0,C 180,E1 -14460.726,E2 -14460.726} C_VEL
LIN {X 0,Y 351.08,Z 348.938,A -85,B 0,C 180,E1 -14461.245,E2 -14461.245} C_VEL
LIN {X 0,Y 349.598,Z 363.846,A -85,B 0,C 180,E1 -14461.971,E2 -14461.971} C_VEL
LIN {X 0,Y 347.937,Z 378.869,A -85,B 0,C 180,E1 -14462.974,E2 -14462.974} C_VEL
LIN {X 0,Y 346.061,Z 392.261,A -85,B 0,C 180,E1 -14464.111,E2 -14464.111} C_VEL
LIN {X 0,Y 343.988,Z 404.67,A -85,B 0,C 180,E1 -14465.4,E2 -14465.4} C_VEL
LIN {X 0,Y 341.757,Z 417.293,A -85,B 0,C 180,E1 -14467,E2 -14467} C_VEL
LIN {X 0,Y 339.694,Z 428.503,A -85,B 0,C 180,E1 -14468.727,E2 -14468.727} C_VEL
LIN {X 0,Y 337.847,Z 438.411,A -85,B 0,C 180,E1 -14470.559,E2 -14470.559} C_VEL
LIN {X 0,Y 336.084,Z 447.889,A -85,B 0,C 180,E1 -14472.663,E2 -14472.663} C_VEL
LIN {X 0,Y 334.651,Z 455.986,A -85,B 0,C 180,E1 -14474.843,E2 -14474.843} C_VEL
LIN {X 0,Y 333.545,Z 463.155,A -85,B 0,C 180,E1 -14477.218,E2 -14477.218} C_VEL
LIN {X 0,Y 332.673,Z 469,A -85,B 0,C 180,E1 -14479.655,E2 -14479.655} C_VEL
LIN {X 0,Y 332.32,Z 472.475,A -85,B 0,C 180,E1 -14481.487,E2 -14481.487} C_VEL
LIN {X 0,Y 332.018,Z 476.309,A -85,B 0,C 180,E1 -14484.195,E2 -14484.195} C_VEL
LIN {X 0,Y 331.935,Z 478.294,A -85,B 0,C 180,E1 -14486.358,E2 -14486.358} C_VEL
LIN {X 0,Y 331.861,Z 479.453,A -85,B 0,C 180,E1 -14488.786,E2 -14488.786} C_VEL
LIN {X 0,Y 331.861,Z 479.45,A -85,B 0,C 180,E1 -14491.213,E2 -14491.213} C_VEL
LIN {X 0,Y 331.935,Z 478.279,A -85,B 0,C 180,E1 -14493.642,E2 -14493.642} C_VEL
LIN {X 0,Y 332.04,Z 475.962,A -85,B 0,C 180,E1 -14496.075,E2 -14496.075} C_VEL
LIN {X 0,Y 332.32,Z 472.448,A -85,B 0,C 180,E1 -14498.513,E2 -14498.513} C_VEL
LIN {X 0,Y 332.805,Z 467.648,A -85,B 0,C 180,E1 -14500.956,E2 -14500.956} C_VEL
LIN {X 0,Y 333.758,Z 461.433,A -85,B 0,C 180,E1 -14503.393,E2 -14503.393} C_VEL
LIN {X 0,Y 335.024,Z 453.626,A -85,B 0,C 180,E1 -14505.826,E2 -14505.826} C_VEL
LIN {X 0,Y 336.547,Z 445.324,A -85,B 0,C 180,E1 -14507.94,E2 -14507.94} C_VEL
LIN {X 0,Y 338.192,Z 436.839,A -85,B 0,C 180,E1 -14509.736,E2 -14509.736} C_VEL
LIN {X 0,Y 340.064,Z 426.196,A -85,B 0,C 180,E1 -14511.641,E2 -14511.641} C_VEL
LIN {X 0,Y 342.151,Z 415.033,A -85,B 0,C 180,E1 -14513.291,E2 -14513.291} C_VEL
LIN {X 0,Y 344.16,Z 403.231,A -85,B 0,C 180,E1 -14514.748,E2 -14514.748} C_VEL
LIN {X 0,Y 346.228,Z 390.481,A -85,B 0,C 180,E1 -14516.038,E2 -14516.038} C_VEL
LIN {X 0,Y 348.201,Z 376.261,A -85,B 0,C 180,E1 -14517.197,E2 -14517.197} C_VEL
LIN {X 0,Y 349.744,Z 362.236,A -85,B 0,C 180,E1 -14518.097,E2 -14518.097} C_VEL
LIN {X 0,Y 351.053,Z 348.503,A -85,B 0,C 180,E1 -14518.757,E2 -14518.757} C_VEL
LIN {X 0,Y 352.097,Z 332.753,A -85,B 0,C 180,E1 -14519.277,E2 -14519.277} C_VEL
LIN {X 0,Y 355.47,Z 219.42,A -85,B 0,C 180,E1 -14521.596,E2 -14521.596} C_VEL
LIN {X 0,Y 355.534,Z 212.459,A -85,B 0,C 180,E1 -14521.752,E2 -14521.752} C_VEL
LIN {X 0,Y 353.421,Z 202.002,A -85,B 0,C 180,E1 -14522.208,E2 -14522.208} C_VEL
LIN {X 0,Y 345.726,Z 184.765,A -85,B 0,C 180,E1 -14523.432,E2 -14523.432} C_VEL
LIN {X 0,Y 337.478,Z 168.042,A -85,B 0,C 180,E1 -14524.813,E2 -14524.813} C_VEL
LIN {X 0,Y 334.422,Z 157.151,A -85,B 0,C 180,E1 -14527.856,E2 -14527.856} C_VEL
LIN {X 0,Y 333.667,Z 154.601,A -85,B 0,C 180,E1 -14528.671,E2 -14528.671} C_VEL
LIN {X 0,Y 333.632,Z 154.537,A -85,B 0,C 180,E1 -14532.5,E2 -14532.5} C_VEL
LIN {X 0,Y 333.596,Z 154.553,A -85,B 0,C 180,E1 -14535.955,E2 -14535.955} C_VEL
LIN {X 0,Y 333.647,Z 154.514,A -85,B 0,C 180,E1 -14539.316,E2 -14539.316} C_VEL
LIN {X 0,Y 333.665,Z 154.549,A -85,B 0,C 180,E1 -14543.168,E2 -14543.168} C_VEL
LIN {X 0,Y 333.674,Z 154.508,A -85,B 0,C 180,E1 -14545.341,E2 -14545.341} C_VEL
LIN {X 0,Y 333.703,Z 154.526,A -85,B 0,C 180,E1 -14549.71,E2 -14549.71} C_VEL
LIN {X 0,Y 333.744,Z 154.535,A -85,B 0,C 180,E1 -14552.401,E2 -14552.401} C_VEL
LIN {X 0,Y 333.728,Z 154.531,A -85,B 0,C 180,E1 -14555.091,E2 -14555.091} C_VEL
LIN {X 0,Y 333.68,Z 154.529,A -85,B 0,C 180,E1 -14559.019,E2 -14559.019} C_VEL
LIN {X 0,Y 333.795,Z 154.531,A -85,B 0,C 180,E1 -14561.59,E2 -14561.59} C_VEL
LIN {X 0,Y 333.809,Z 154.518,A -85,B 0,C 180,E1 -14565.577,E2 -14565.577} C_VEL
LIN {X 0,Y 333.819,Z 154.516,A -85,B 0,C 180,E1 -14569.078,E2 -14569.078} C_VEL
LIN {X 0,Y 333.964,Z 154.508,A -85,B 0,C 180,E1 -14572.746,E2 -14572.746} C_VEL
LIN {X 0,Y 333.798,Z 154.516,A -85,B 0,C 180,E1 -14575.169,E2 -14575.169} C_VEL
LIN {X 0,Y 334.102,Z 154.48,A -85,B 0,C 180,E1 -14577.589,E2 -14577.589} C_VEL
LIN {X 0,Y 334.208,Z 154.477,A -85,B 0,C 180,E1 -14580,E2 -14580} C_VEL
LIN {X 0,Y 334.073,Z 154.475,A -85,B 0,C 180,E1 -14582.412,E2 -14582.412} C_VEL
LIN {X 0,Y 333.97,Z 154.504,A -85,B 0,C 180,E1 -14586.491,E2 -14586.491} C_VEL
LIN {X 0,Y 333.822,Z 154.515,A -85,B 0,C 180,E1 -14589.696,E2 -14589.696} C_VEL
LIN {X 0,Y 333.794,Z 154.519,A -85,B 0,C 180,E1 -14593.392,E2 -14593.392} C_VEL
LIN {X 0,Y 333.719,Z 154.539,A -85,B 0,C 180,E1 -14597.148,E2 -14597.148} C_VEL
LIN {X 0,Y 333.672,Z 154.53,A -85,B 0,C 180,E1 -14599.694,E2 -14599.694} C_VEL
LIN {X 0,Y 333.646,Z 154.546,A -85,B 0,C 180,E1 -14603.592,E2 -14603.592} C_VEL
LIN {X 0,Y 333.667,Z 154.548,A -85,B 0,C 180,E1 -14607.606,E2 -14607.606} C_VEL
LIN {X 0,Y 333.656,Z 154.513,A -85,B 0,C 180,E1 -14610.366,E2 -14610.366} C_VEL
LIN {X 0,Y 333.637,Z 154.5,A -85,B 0,C 180,E1 -14613.209,E2 -14613.209} C_VEL
LIN {X 0,Y 333.676,Z 154.548,A -85,B 0,C 180,E1 -14616.139,E2 -14616.139} C_VEL
LIN {X 0,Y 333.602,Z 154.516,A -85,B 0,C 180,E1 -14619.199,E2 -14619.199} C_VEL
LIN {X 0,Y 333.629,Z 154.541,A -85,B 0,C 180,E1 -14622.499,E2 -14622.499} C_VEL
LIN {X 0,Y 333.594,Z 154.533,A -85,B 0,C 180,E1 -14625.955,E2 -14625.955} C_VEL
LIN {X 0,Y 333.602,Z 154.543,A -85,B 0,C 180,E1 -14629.325,E2 -14629.325} C_VEL
LIN {X 0,Y 333.695,Z 154.679,A -85,B 0,C 180,E1 -14632.584,E2 -14632.584} C_VEL
LIN {X 0,Y 336.018,Z 162.835,A -85,B 0,C 180,E1 -14635.033,E2 -14635.033} C_VEL
LIN {X 0,Y 339.034,Z 168.811,A -85,B 0,C 180,E1 -14635.597,E2 -14635.597} C_VEL
LIN {X 0,Y 348.287,Z 187.397,A -85,B 0,C 180,E1 -14637.085,E2 -14637.085} C_VEL
LIN {X 0,Y 355.672,Z 204.34,A -85,B 0,C 180,E1 -14638.25,E2 -14638.25} C_VEL
LIN {X 0,Y 355.762,Z 208.977,A -85,B 0,C 180,E1 -14638.367,E2 -14638.367} C_VEL
LIN {X 0,Y 352.248,Z 326.86,A -85,B 0,C 180,E1 -14640.778,E2 -14640.778} C_VEL
LIN {X 0,Y 351.3,Z 341.739,A -85,B 0,C 180,E1 -14641.265,E2 -14641.265} C_VEL
LIN {X 0,Y 350.078,Z 355.489,A -85,B 0,C 180,E1 -14641.916,E2 -14641.916} C_VEL
LIN {X 0,Y 348.49,Z 370.223,A -85,B 0,C 180,E1 -14642.853,E2 -14642.853} C_VEL
LIN {X 0,Y 346.607,Z 384.223,A -85,B 0,C 180,E1 -14643.993,E2 -14643.993} C_VEL
LIN {X 0,Y 344.602,Z 397.023,A -85,B 0,C 180,E1 -14645.286,E2 -14645.286} C_VEL
LIN {X 0,Y 342.363,Z 409.921,A -85,B 0,C 180,E1 -14646.884,E2 -14646.884} C_VEL
LIN {X 0,Y 340.472,Z 420.756,A -85,B 0,C 180,E1 -14648.516,E2 -14648.516} C_VEL
LIN {X 0,Y 338.548,Z 430.674,A -85,B 0,C 180,E1 -14650.285,E2 -14650.285} C_VEL
LIN {X 0,Y 336.722,Z 440.413,A -85,B 0,C 180,E1 -14652.384,E2 -14652.384} C_VEL
LIN {X 0,Y 335.166,Z 448.629,A -85,B 0,C 180,E1 -14654.523,E2 -14654.523} C_VEL
LIN {X 0,Y 334.144,Z 455.229,A -85,B 0,C 180,E1 -14656.623,E2 -14656.623} C_VEL
LIN {X 0,Y 333.072,Z 461.434,A -85,B 0,C 180,E1 -14659.053,E2 -14659.053} C_VEL
LIN {X 0,Y 332.466,Z 466.225,A -85,B 0,C 180,E1 -14661.491,E2 -14661.491} C_VEL
LIN {X 0,Y 332.135,Z 469.826,A -85,B 0,C 180,E1 -14664.003,E2 -14664.003} C_VEL
LIN {X 0,Y 331.997,Z 472.057,A -85,B 0,C 180,E1 -14666.359,E2 -14666.359} C_VEL
LIN {X 0,Y 331.873,Z 473.243,A -85,B 0,C 180,E1 -14668.787,E2 -14668.787} C_VEL
LIN {X 0,Y 331.874,Z 473.258,A -85,B 0,C 180,E1 -14671.213,E2 -14671.213} C_VEL
LIN {X 0,Y 331.994,Z 472.131,A -85,B 0,C 180,E1 -14673.641,E2 -14673.641} C_VEL
LIN {X 0,Y 332.098,Z 469.867,A -85,B 0,C 180,E1 -14676.074,E2 -14676.074} C_VEL
LIN {X 0,Y 332.46,Z 466.409,A -85,B 0,C 180,E1 -14678.51,E2 -14678.51} C_VEL
LIN {X 0,Y 333.042,Z 461.677,A -85,B 0,C 180,E1 -14680.948,E2 -14680.948} C_VEL
LIN {X 0,Y 334.087,Z 455.545,A -85,B 0,C 180,E1 -14683.38,E2 -14683.38} C_VEL
LIN {X 0,Y 335.33,Z 447.828,A -85,B 0,C 180,E1 -14685.811,E2 -14685.811} C_VEL
LIN {X 0,Y 336.876,Z 439.601,A -85,B 0,C 180,E1 -14687.922,E2 -14687.922} C_VEL
LIN {X 0,Y 338.791,Z 429.691,A -85,B 0,C 180,E1 -14690.016,E2 -14690.016} C_VEL
LIN {X 0,Y 340.362,Z 421.115,A -85,B 0,C 180,E1 -14691.536,E2 -14691.536} C_VEL
LIN {X 0,Y 342.495,Z 409.575,A -85,B 0,C 180,E1 -14693.267,E2 -14693.267} C_VEL
LIN {X 0,Y 344.707,Z 396.604,A -85,B 0,C 180,E1 -14694.867,E2 -14694.867} C_VEL
LIN {X 0,Y 346.712,Z 383.721,A -85,B 0,C 180,E1 -14696.16,E2 -14696.16} C_VEL
LIN {X 0,Y 348.543,Z 370.33,A -85,B 0,C 180,E1 -14697.245,E2 -14697.245} C_VEL
LIN {X 0,Y 350.071,Z 355.804,A -85,B 0,C 180,E1 -14698.175,E2 -14698.175} C_VEL
LIN {X 0,Y 351.104,Z 344.769,A -85,B 0,C 180,E1 -14698.717,E2 -14698.717} C_VEL
LIN {X 0,Y 350.873,Z 339.135,A -85,B 0,C 180,E1 -14699.013,E2 -14699.013} C_VEL
LIN {X 0,Y 347.171,Z 322.568,A -85,B 0,C 180,E1 -14699.925,E2 -14699.925} C_VEL
LIN {X 0,Y 346.54,Z 316.83,A -85,B 0,C 180,E1 -14700.128,E2 -14700.128} C_VEL
LIN {X 0,Y 346.552,Z 314.881,A -85,B 0,C 180,E1 -14700.173,E2 -14700.173} C_VEL
LIN {X 0,Y 349.831,Z 206.858,A -85,B 0,C 180,E1 -14702.399,E2 -14702.399} C_VEL
LIN {X 0,Y 341.894,Z 188.68,A -85,B 0,C 180,E1 -14703.697,E2 -14703.697} C_VEL
LIN {X 0,Y 332.855,Z 170.706,A -85,B 0,C 180,E1 -14705.207,E2 -14705.207} C_VEL
LIN {X 0,Y 328.746,Z 162.972,A -85,B 0,C 180,E1 -14705.966,E2 -14705.966} C_VEL
LIN {X 0,Y 326.62,Z 155.598,A -85,B 0,C 180,E1 -14708.253,E2 -14708.253} C_VEL
LIN {X 0,Y 326.561,Z 155.434,A -85,B 0,C 180,E1 -14711.848,E2 -14711.848} C_VEL
LIN {X 0,Y 326.525,Z 155.42,A -85,B 0,C 180,E1 -14715.258,E2 -14715.258} C_VEL
LIN {X 0,Y 326.561,Z 155.408,A -85,B 0,C 180,E1 -14718.152,E2 -14718.152} C_VEL
LIN {X 0,Y 326.568,Z 155.398,A -85,B 0,C 180,E1 -14721.383,E2 -14721.383} C_VEL
LIN {X 0,Y 326.621,Z 155.417,A -85,B 0,C 180,E1 -14724.851,E2 -14724.851} C_VEL
LIN {X 0,Y 326.608,Z 155.37,A -85,B 0,C 180,E1 -14727.455,E2 -14727.455} C_VEL
LIN {X 0,Y 326.616,Z 155.403,A -85,B 0,C 180,E1 -14730.336,E2 -14730.336} C_VEL
LIN {X 0,Y 326.602,Z 155.411,A -85,B 0,C 180,E1 -14734.509,E2 -14734.509} C_VEL
LIN {X 0,Y 326.616,Z 155.418,A -85,B 0,C 180,E1 -14738.543,E2 -14738.543} C_VEL
LIN {X 0,Y 326.655,Z 155.421,A -85,B 0,C 180,E1 -14742.469,E2 -14742.469} C_VEL
LIN {X 0,Y 326.757,Z 155.391,A -85,B 0,C 180,E1 -14746.314,E2 -14746.314} C_VEL
LIN {X 0,Y 326.785,Z 155.393,A -85,B 0,C 180,E1 -14750.093,E2 -14750.093} C_VEL
LIN {X 0,Y 326.954,Z 155.381,A -85,B 0,C 180,E1 -14753.83,E2 -14753.83} C_VEL
LIN {X 0,Y 327.015,Z 155.353,A -85,B 0,C 180,E1 -14757.536,E2 -14757.536} C_VEL
LIN {X 0,Y 327.142,Z 155.358,A -85,B 0,C 180,E1 -14760,E2 -14760} C_VEL
LIN {X 0,Y 327.037,Z 155.359,A -85,B 0,C 180,E1 -14762.463,E2 -14762.463} C_VEL
LIN {X 0,Y 326.952,Z 155.381,A -85,B 0,C 180,E1 -14766.17,E2 -14766.17} C_VEL
LIN {X 0,Y 326.785,Z 155.384,A -85,B 0,C 180,E1 -14769.907,E2 -14769.907} C_VEL
LIN {X 0,Y 326.761,Z 155.402,A -85,B 0,C 180,E1 -14773.685,E2 -14773.685} C_VEL
LIN {X 0,Y 326.701,Z 155.414,A -85,B 0,C 180,E1 -14777.528,E2 -14777.528} C_VEL
LIN {X 0,Y 326.659,Z 155.408,A -85,B 0,C 180,E1 -14780.135,E2 -14780.135} C_VEL
LIN {X 0,Y 326.65,Z 155.421,A -85,B 0,C 180,E1 -14784.129,E2 -14784.129} C_VEL
LIN {X 0,Y 326.686,Z 155.404,A -85,B 0,C 180,E1 -14786.857,E2 -14786.857} C_VEL
LIN {X 0,Y 326.64,Z 155.399,A -85,B 0,C 180,E1 -14790.611,E2 -14790.611} C_VEL
LIN {X 0,Y 326.607,Z 155.377,A -85,B 0,C 180,E1 -14794.019,E2 -14794.019} C_VEL
LIN {X 0,Y 326.628,Z 155.424,A -85,B 0,C 180,E1 -14797.238,E2 -14797.238} C_VEL
LIN {X 0,Y 326.577,Z 155.396,A -85,B 0,C 180,E1 -14801.131,E2 -14801.131} C_VEL
LIN {X 0,Y 326.527,Z 155.42,A -85,B 0,C 180,E1 -14804.743,E2 -14804.743} C_VEL
LIN {X 0,Y 326.576,Z 155.429,A -85,B 0,C 180,E1 -14808.154,E2 -14808.154} C_VEL
LIN {X 0,Y 326.642,Z 155.602,A -85,B 0,C 180,E1 -14810.629,E2 -14810.629} C_VEL
LIN {X 0,Y 329.372,Z 165.03,A -85,B 0,C 180,E1 -14813.486,E2 -14813.486} C_VEL
LIN {X 0,Y 330.241,Z 168.131,A -85,B 0,C 180,E1 -14814.293,E2 -14814.293} C_VEL
LIN {X 0,Y 338.203,Z 183.719,A -85,B 0,C 180,E1 -14815.673,E2 -14815.673} C_VEL
LIN {X 0,Y 347.427,Z 203.993,A -85,B 0,C 180,E1 -14817.193,E2 -14817.193} C_VEL
LIN {X 0,Y 348.509,Z 207.763,A -85,B 0,C 180,E1 -14817.398,E2 -14817.398} C_VEL
LIN {X 0,Y 349.679,Z 215.585,A -85,B 0,C 180,E1 -14817.706,E2 -14817.706} C_VEL
LIN {X 0,Y 345.953,Z 333.448,A -85,B 0,C 180,E1 -14820.151,E2 -14820.151} C_VEL
LIN {X 0,Y 344.867,Z 348.882,A -85,B 0,C 180,E1 -14820.677,E2 -14820.677} C_VEL
LIN {X 0,Y 343.333,Z 363.787,A -85,B 0,C 180,E1 -14821.413,E2 -14821.413} C_VEL
LIN {X 0,Y 341.652,Z 378.537,A -85,B 0,C 180,E1 -14822.412,E2 -14822.412} C_VEL
LIN {X 0,Y 339.66,Z 392.198,A -85,B 0,C 180,E1 -14823.585,E2 -14823.585} C_VEL
LIN {X 0,Y 337.493,Z 404.607,A -85,B 0,C 180,E1 -14824.894,E2 -14824.894} C_VEL
LIN {X 0,Y 335.177,Z 417.23,A -85,B 0,C 180,E1 -14826.522,E2 -14826.522} C_VEL
LIN {X 0,Y 332.884,Z 429.186,A -85,B 0,C 180,E1 -14828.406,E2 -14828.406} C_VEL
LIN {X 0,Y 331.137,Z 438.347,A -85,B 0,C 180,E1 -14830.149,E2 -14830.149} C_VEL
LIN {X 0,Y 329.239,Z 447.824,A -85,B 0,C 180,E1 -14832.291,E2 -14832.291} C_VEL
LIN {X 0,Y 327.787,Z 455.721,A -85,B 0,C 180,E1 -14834.455,E2 -14834.455} C_VEL
LIN {X 0,Y 326.563,Z 463.089,A -85,B 0,C 180,E1 -14836.94,E2 -14836.94} C_VEL
LIN {X 0,Y 325.648,Z 468.934,A -85,B 0,C 180,E1 -14839.43,E2 -14839.43} C_VEL
LIN {X 0,Y 325.272,Z 472.409,A -85,B 0,C 180,E1 -14841.301,E2 -14841.301} C_VEL
LIN {X 0,Y 324.956,Z 475.92,A -85,B 0,C 180,E1 -14843.792,E2 -14843.792} C_VEL
LIN {X 0,Y 324.843,Z 478.228,A -85,B 0,C 180,E1 -14846.279,E2 -14846.279} C_VEL
LIN {X 0,Y 324.772,Z 479.387,A -85,B 0,C 180,E1 -14848.76,E2 -14848.76} C_VEL
LIN {X 0,Y 324.772,Z 479.384,A -85,B 0,C 180,E1 -14851.24,E2 -14851.24} C_VEL
LIN {X 0,Y 324.844,Z 478.213,A -85,B 0,C 180,E1 -14853.721,E2 -14853.721} C_VEL
LIN {X 0,Y 324.956,Z 475.895,A -85,B 0,C 180,E1 -14856.208,E2 -14856.208} C_VEL
LIN {X 0,Y 325.271,Z 472.381,A -85,B 0,C 180,E1 -14858.699,E2 -14858.699} C_VEL
LIN {X 0,Y 325.783,Z 467.58,A -85,B 0,C 180,E1 -14861.195,E2 -14861.195} C_VEL
LIN {X 0,Y 326.778,Z 461.364,A -85,B 0,C 180,E1 -14863.685,E2 -14863.685} C_VEL
LIN {X 0,Y 328.116,Z 453.558,A -85,B 0,C 180,E1 -14866.168,E2 -14866.168} C_VEL
LIN {X 0,Y 329.72,Z 445.255,A -85,B 0,C 180,E1 -14868.324,E2 -14868.324} C_VEL
LIN {X 0,Y 331.801,Z 435.251,A -85,B 0,C 180,E1 -14870.456,E2 -14870.456} C_VEL
LIN {X 0,Y 333.682,Z 425.018,A -85,B 0,C 180,E1 -14872.279,E2 -14872.279} C_VEL
LIN {X 0,Y 336.025,Z 412.82,A -85,B 0,C 180,E1 -14874.07,E2 -14874.07} C_VEL
LIN {X 0,Y 338.166,Z 400.574,A -85,B 0,C 180,E1 -14875.546,E2 -14875.546} C_VEL
LIN {X 0,Y 340.354,Z 387.242,A -85,B 0,C 180,E1 -14876.853,E2 -14876.853} C_VEL
LIN {X 0,Y 342.151,Z 374.007,A -85,B 0,C 180,E1 -14877.901,E2 -14877.901} C_VEL
LIN {X 0,Y 343.757,Z 359.562,A -85,B 0,C 180,E1 -14878.798,E2 -14878.798} C_VEL
LIN {X 0,Y 345.126,Z 344.76,A -85,B 0,C 180,E1 -14879.466,E2 -14879.466} C_VEL
LIN {X 0,Y 346.07,Z 329.656,A -85,B 0,C 180,E1 -14879.922,E2 -14879.922} C_VEL
LIN {X 0,Y 349.579,Z 215.155,A -85,B 0,C 180,E1 -14882.291,E2 -14882.291} C_VEL
LIN {X 0,Y 348.632,Z 208.733,A -85,B 0,C 180,E1 -14882.543,E2 -14882.543} C_VEL
LIN {X 0,Y 347.592,Z 204.476,A -85,B 0,C 180,E1 -14882.754,E2 -14882.754} C_VEL
LIN {X 0,Y 339.454,Z 186.372,A -85,B 0,C 180,E1 -14884.091,E2 -14884.091} C_VEL
LIN {X 0,Y 331.899,Z 171.396,A -85,B 0,C 180,E1 -14885.363,E2 -14885.363} C_VEL
LIN {X 0,Y 330.122,Z 167.787,A -85,B 0,C 180,E1 -14885.73,E2 -14885.73} C_VEL
LIN {X 0,Y 327.403,Z 158.268,A -85,B 0,C 180,E1 -14888.5,E2 -14888.5} C_VEL
LIN {X 0,Y 326.615,Z 155.498,A -85,B 0,C 180,E1 -14889.392,E2 -14889.392} C_VEL
LIN {X 0,Y 326.561,Z 155.406,A -85,B 0,C 180,E1 -14893.526,E2 -14893.526} C_VEL
LIN {X 0,Y 326.576,Z 155.428,A -85,B 0,C 180,E1 -14897.028,E2 -14897.028} C_VEL
LIN {X 0,Y 326.611,Z 155.398,A -85,B 0,C 180,E1 -14900.773,E2 -14900.773} C_VEL
LIN {X 0,Y 326.612,Z 155.406,A -85,B 0,C 180,E1 -14904.48,E2 -14904.48} C_VEL
LIN {X 0,Y 326.608,Z 155.371,A -85,B 0,C 180,E1 -14907.456,E2 -14907.456} C_VEL
LIN {X 0,Y 326.661,Z 155.415,A -85,B 0,C 180,E1 -14910.341,E2 -14910.341} C_VEL
LIN {X 0,Y 326.691,Z 155.402,A -85,B 0,C 180,E1 -14914.516,E2 -14914.516} C_VEL
LIN {X 0,Y 326.646,Z 155.406,A -85,B 0,C 180,E1 -14918.545,E2 -14918.545} C_VEL
LIN {X 0,Y 326.745,Z 155.409,A -85,B 0,C 180,E1 -14921.178,E2 -14921.178} C_VEL
LIN {X 0,Y 326.764,Z 155.393,A -85,B 0,C 180,E1 -14925.433,E2 -14925.433} C_VEL
LIN {X 0,Y 326.76,Z 155.397,A -85,B 0,C 180,E1 -14928.839,E2 -14928.839} C_VEL
LIN {X 0,Y 326.919,Z 155.383,A -85,B 0,C 180,E1 -14932.589,E2 -14932.589} C_VEL
LIN {X 0,Y 326.765,Z 155.393,A -85,B 0,C 180,E1 -14935.065,E2 -14935.065} C_VEL
LIN {X 0,Y 327.043,Z 155.358,A -85,B 0,C 180,E1 -14937.537,E2 -14937.537} C_VEL
LIN {X 0,Y 327.16,Z 155.355,A -85,B 0,C 180,E1 -14940,E2 -14940} C_VEL
LIN {X 0,Y 327.017,Z 155.353,A -85,B 0,C 180,E1 -14942.464,E2 -14942.464} C_VEL
LIN {X 0,Y 326.931,Z 155.38,A -85,B 0,C 180,E1 -14946.479,E2 -14946.479} C_VEL
LIN {X 0,Y 326.784,Z 155.393,A -85,B 0,C 180,E1 -14949.907,E2 -14949.907} C_VEL
LIN {X 0,Y 326.758,Z 155.392,A -85,B 0,C 180,E1 -14953.686,E2 -14953.686} C_VEL
LIN {X 0,Y 326.665,Z 155.419,A -85,B 0,C 180,E1 -14957.53,E2 -14957.53} C_VEL
LIN {X 0,Y 326.615,Z 155.417,A -85,B 0,C 180,E1 -14961.457,E2 -14961.457} C_VEL
LIN {X 0,Y 326.602,Z 155.411,A -85,B 0,C 180,E1 -14965.491,E2 -14965.491} C_VEL
LIN {X 0,Y 326.615,Z 155.405,A -85,B 0,C 180,E1 -14969.664,E2 -14969.664} C_VEL
LIN {X 0,Y 326.617,Z 155.37,A -85,B 0,C 180,E1 -14972.946,E2 -14972.946} C_VEL
LIN {X 0,Y 326.613,Z 155.42,A -85,B 0,C 180,E1 -14975.52,E2 -14975.52} C_VEL
LIN {X 0,Y 326.572,Z 155.39,A -85,B 0,C 180,E1 -14979.218,E2 -14979.218} C_VEL
LIN {X 0,Y 326.574,Z 155.428,A -85,B 0,C 180,E1 -14982.971,E2 -14982.971} C_VEL
LIN {X 0,Y 326.572,Z 155.414,A -85,B 0,C 180,E1 -14987.029,E2 -14987.029} C_VEL
LIN {X 0,Y 326.597,Z 155.418,A -85,B 0,C 180,E1 -14991.388,E2 -14991.388} C_VEL
LIN {X 0,Y 326.649,Z 155.735,A -85,B 0,C 180,E1 -14991.938,E2 -14991.938} C_VEL
LIN {X 0,Y 328.834,Z 163.146,A -85,B 0,C 180,E1 -14994.186,E2 -14994.186} C_VEL
LIN {X 0,Y 335.935,Z 176.677,A -85,B 0,C 180,E1 -14995.433,E2 -14995.433} C_VEL
LIN {X 0,Y 343.761,Z 192.831,A -85,B 0,C 180,E1 -14996.727,E2 -14996.727} C_VEL
LIN {X 0,Y 349.768,Z 206.716,A -85,B 0,C 180,E1 -14997.704,E2 -14997.704} C_VEL
LIN {X 0,Y 346.528,Z 313.809,A -85,B 0,C 180,E1 -14999.912,E2 -14999.912} C_VEL
LIN {X 0,Y 345.693,Z 332.974,A -85,B 0,C 180,E1 -15000.378,E2 -15000.378} C_VEL
LIN {X 0,Y 344.565,Z 347.925,A -85,B 0,C 180,E1 -15000.967,E2 -15000.967} C_VEL
LIN {X 0,Y 343.072,Z 362.988,A -85,B 0,C 180,E1 -15001.808,E2 -15001.808} C_VEL
LIN {X 0,Y 341.211,Z 377.749,A -85,B 0,C 180,E1 -15002.895,E2 -15002.895} C_VEL
LIN {X 0,Y 339.015,Z 391.716,A -85,B 0,C 180,E1 -15004.193,E2 -15004.193} C_VEL
LIN {X 0,Y 336.871,Z 404.44,A -85,B 0,C 180,E1 -15005.667,E2 -15005.667} C_VEL
LIN {X 0,Y 334.796,Z 415.508,A -85,B 0,C 180,E1 -15007.213,E2 -15007.213} C_VEL
LIN {X 0,Y 332.855,Z 425.962,A -85,B 0,C 180,E1 -15008.965,E2 -15008.965} C_VEL
LIN {X 0,Y 330.99,Z 435.161,A -85,B 0,C 180,E1 -15010.785,E2 -15010.785} C_VEL
LIN {X 0,Y 329.173,Z 444.158,A -85,B 0,C 180,E1 -15012.928,E2 -15012.928} C_VEL
LIN {X 0,Y 327.733,Z 451.615,A -85,B 0,C 180,E1 -15015.088,E2 -15015.088} C_VEL
LIN {X 0,Y 326.894,Z 456.977,A -85,B 0,C 180,E1 -15016.953,E2 -15016.953} C_VEL
LIN {X 0,Y 325.881,Z 462.828,A -85,B 0,C 180,E1 -15019.437,E2 -15019.437} C_VEL
LIN {X 0,Y 325.427,Z 466.293,A -85,B 0,C 180,E1 -15021.305,E2 -15021.305} C_VEL
LIN {X 0,Y 325.024,Z 470.131,A -85,B 0,C 180,E1 -15024.076,E2 -15024.076} C_VEL
LIN {X 0,Y 324.903,Z 472.124,A -85,B 0,C 180,E1 -15026.279,E2 -15026.279} C_VEL
LIN {X 0,Y 324.785,Z 473.309,A -85,B 0,C 180,E1 -15028.76,E2 -15028.76} C_VEL
LIN {X 0,Y 324.785,Z 473.324,A -85,B 0,C 180,E1 -15031.24,E2 -15031.24} C_VEL
LIN {X 0,Y 324.9,Z 472.197,A -85,B 0,C 180,E1 -15033.721,E2 -15033.721} C_VEL
LIN {X 0,Y 325.008,Z 469.933,A -85,B 0,C 180,E1 -15036.207,E2 -15036.207} C_VEL
LIN {X 0,Y 325.421,Z 466.475,A -85,B 0,C 180,E1 -15038.695,E2 -15038.695} C_VEL
LIN {X 0,Y 326.02,Z 461.742,A -85,B 0,C 180,E1 -15041.187,E2 -15041.187} C_VEL
LIN {X 0,Y 327.134,Z 455.61,A -85,B 0,C 180,E1 -15043.669,E2 -15043.669} C_VEL
LIN {X 0,Y 328.455,Z 447.893,A -85,B 0,C 180,E1 -15046.151,E2 -15046.151} C_VEL
LIN {X 0,Y 330.077,Z 439.665,A -85,B 0,C 180,E1 -15048.304,E2 -15048.304} C_VEL
LIN {X 0,Y 332.113,Z 429.755,A -85,B 0,C 180,E1 -15050.436,E2 -15050.436} C_VEL
LIN {X 0,Y 334.019,Z 419.597,A -85,B 0,C 180,E1 -15052.255,E2 -15052.255} C_VEL
LIN {X 0,Y 336.357,Z 407.503,A -85,B 0,C 180,E1 -15054.044,E2 -15054.044} C_VEL
LIN {X 0,Y 338.478,Z 395.378,A -85,B 0,C 180,E1 -15055.521,E2 -15055.521} C_VEL
LIN {X 0,Y 340.579,Z 382.202,A -85,B 0,C 180,E1 -15056.834,E2 -15056.834} C_VEL
LIN {X 0,Y 342.523,Z 368.248,A -85,B 0,C 180,E1 -15057.943,E2 -15057.943} C_VEL
LIN {X 0,Y 344.032,Z 353.66,A -85,B 0,C 180,E1 -15058.856,E2 -15058.856} C_VEL
LIN {X 0,Y 345.366,Z 338.758,A -85,B 0,C 180,E1 -15059.527,E2 -15059.527} C_VEL
LIN {X 0,Y 346.254,Z 323.44,A -85,B 0,C 180,E1 -15059.988,E2 -15059.988} C_VEL
LIN {X 0,Y 346.552,Z 314.881,A -85,B 0,C 180,E1 -15060.173,E2 -15060.173} C_VEL
LIN {X 0,Y 346.204,Z 309.074,A -85,B 0,C 180,E1 -15060.343,E2 -15060.343} C_VEL
LIN {X 0,Y 341.806,Z 290.442,A -85,B 0,C 180,E1 -15061.224,E2 -15061.224} C_VEL
LIN {X 0,Y 341.435,Z 284.635,A -85,B 0,C 180,E1 -15061.401,E2 -15061.401} C_VEL
LIN {X 0,Y 343.791,Z 208.787,A -85,B 0,C 180,E1 -15062.994,E2 -15062.994} C_VEL
LIN {X 0,Y 335.35,Z 189.637,A -85,B 0,C 180,E1 -15064.423,E2 -15064.423} C_VEL
LIN {X 0,Y 327.537,Z 174.296,A -85,B 0,C 180,E1 -15065.772,E2 -15065.772} C_VEL
LIN {X 0,Y 321.53,Z 163.092,A -85,B 0,C 180,E1 -15066.899,E2 -15066.899} C_VEL
LIN {X 0,Y 319.572,Z 156.494,A -85,B 0,C 180,E1 -15069.014,E2 -15069.014} C_VEL
LIN {X 0,Y 319.55,Z 156.29,A -85,B 0,C 180,E1 -15072.984,E2 -15072.984} C_VEL
LIN {X 0,Y 319.551,Z 156.304,A -85,B 0,C 180,E1 -15077.016,E2 -15077.016} C_VEL
LIN {X 0,Y 319.515,Z 156.264,A -85,B 0,C 180,E1 -15080.366,E2 -15080.366} C_VEL
LIN {X 0,Y 319.581,Z 156.298,A -85,B 0,C 180,E1 -15084.457,E2 -15084.457} C_VEL
LIN {X 0,Y 319.523,Z 156.249,A -85,B 0,C 180,E1 -15088.137,E2 -15088.137} C_VEL
LIN {X 0,Y 319.572,Z 156.299,A -85,B 0,C 180,E1 -15091.604,E2 -15091.604} C_VEL
LIN {X 0,Y 319.529,Z 156.292,A -85,B 0,C 180,E1 -15095.298,E2 -15095.298} C_VEL
LIN {X 0,Y 319.566,Z 156.301,A -85,B 0,C 180,E1 -15098.045,E2 -15098.045} C_VEL
LIN {X 0,Y 319.609,Z 156.295,A -85,B 0,C 180,E1 -15102.07,E2 -15102.07} C_VEL
LIN {X 0,Y 319.731,Z 156.264,A -85,B 0,C 180,E1 -15106.008,E2 -15106.008} C_VEL
LIN {X 0,Y 319.737,Z 156.273,A -85,B 0,C 180,E1 -15109.872,E2 -15109.872} C_VEL
LIN {X 0,Y 319.91,Z 156.257,A -85,B 0,C 180,E1 -15113.694,E2 -15113.694} C_VEL
LIN {X 0,Y 319.962,Z 156.231,A -85,B 0,C 180,E1 -15117.482,E2 -15117.482} C_VEL
LIN {X 0,Y 320.097,Z 156.235,A -85,B 0,C 180,E1 -15120,E2 -15120} C_VEL
LIN {X 0,Y 319.98,Z 156.236,A -85,B 0,C 180,E1 -15122.518,E2 -15122.518} C_VEL
LIN {X 0,Y 319.908,Z 156.258,A -85,B 0,C 180,E1 -15126.306,E2 -15126.306} C_VEL
LIN {X 0,Y 319.737,Z 156.262,A -85,B 0,C 180,E1 -15130.128,E2 -15130.128} C_VEL
LIN {X 0,Y 319.734,Z 156.276,A -85,B 0,C 180,E1 -15133.992,E2 -15133.992} C_VEL
LIN {X 0,Y 319.66,Z 156.291,A -85,B 0,C 180,E1 -15137.927,E2 -15137.927} C_VEL
LIN {X 0,Y 319.603,Z 156.282,A -85,B 0,C 180,E1 -15140.6,E2 -15140.6} C_VEL
LIN {X 0,Y 319.604,Z 156.291,A -85,B 0,C 180,E1 -15144.696,E2 -15144.696} C_VEL
LIN {X 0,Y 319.617,Z 156.298,A -85,B 0,C 180,E1 -15148.411,E2 -15148.411} C_VEL
LIN {X 0,Y 319.533,Z 156.256,A -85,B 0,C 180,E1 -15151.862,E2 -15151.862} C_VEL
LIN {X 0,Y 319.58,Z 156.283,A -85,B 0,C 180,E1 -15155.543,E2 -15155.543} C_VEL
LIN {X 0,Y 319.559,Z 156.269,A -85,B 0,C 180,E1 -15159.668,E2 -15159.668} C_VEL
LIN {X 0,Y 319.522,Z 156.311,A -85,B 0,C 180,E1 -15163.46,E2 -15163.46} C_VEL
LIN {X 0,Y 319.554,Z 156.282,A -85,B 0,C 180,E1 -15167.016,E2 -15167.016} C_VEL
LIN {X 0,Y 319.584,Z 156.52,A -85,B 0,C 180,E1 -15169.864,E2 -15169.864} C_VEL
LIN {X 0,Y 322.305,Z 165.757,A -85,B 0,C 180,E1 -15172.763,E2 -15172.763} C_VEL
LIN {X 0,Y 322.993,Z 168.041,A -85,B 0,C 180,E1 -15173.362,E2 -15173.362} C_VEL
LIN {X 0,Y 331.646,Z 184.656,A -85,B 0,C 180,E1 -15174.921,E2 -15174.921} C_VEL
LIN {X 0,Y 340.175,Z 203.211,A -85,B 0,C 180,E1 -15176.384,E2 -15176.384} C_VEL
LIN {X 0,Y 342.562,Z 209.194,A -85,B 0,C 180,E1 -15176.795,E2 -15176.795} C_VEL
LIN {X 0,Y 343.626,Z 215.335,A -85,B 0,C 180,E1 -15177.061,E2 -15177.061} C_VEL
LIN {X 0,Y 340.504,Z 313.276,A -85,B 0,C 180,E1 -15179.108,E2 -15179.108} C_VEL
LIN {X 0,Y 339.693,Z 335.785,A -85,B 0,C 180,E1 -15179.629,E2 -15179.629} C_VEL
LIN {X 0,Y 338.47,Z 351.188,A -85,B 0,C 180,E1 -15180.196,E2 -15180.196} C_VEL
LIN {X 0,Y 336.853,Z 366.07,A -85,B 0,C 180,E1 -15180.982,E2 -15180.982} C_VEL
LIN {X 0,Y 335.272,Z 379.159,A -85,B 0,C 180,E1 -15181.902,E2 -15181.902} C_VEL
LIN {X 0,Y 333.286,Z 392.136,A -85,B 0,C 180,E1 -15183.04,E2 -15183.04} C_VEL
LIN {X 0,Y 331.056,Z 404.544,A -85,B 0,C 180,E1 -15184.371,E2 -15184.371} C_VEL
LIN {X 0,Y 328.633,Z 417.166,A -85,B 0,C 180,E1 -15186.026,E2 -15186.026} C_VEL
LIN {X 0,Y 326.399,Z 428.289,A -85,B 0,C 180,E1 -15187.8,E2 -15187.8} C_VEL
LIN {X 0,Y 324.423,Z 438.282,A -85,B 0,C 180,E1 -15189.72,E2 -15189.72} C_VEL
LIN {X 0,Y 322.441,Z 447.759,A -85,B 0,C 180,E1 -15191.905,E2 -15191.905} C_VEL
LIN {X 0,Y 320.881,Z 455.653,A -85,B 0,C 180,E1 -15194.111,E2 -15194.111} C_VEL
LIN {X 0,Y 319.592,Z 463.023,A -85,B 0,C 180,E1 -15196.65,E2 -15196.65} C_VEL
LIN {X 0,Y 318.607,Z 468.868,A -85,B 0,C 180,E1 -15199.193,E2 -15199.193} C_VEL
LIN {X 0,Y 318.2,Z 472.343,A -85,B 0,C 180,E1 -15201.106,E2 -15201.106} C_VEL
LIN {X 0,Y 317.882,Z 475.854,A -85,B 0,C 180,E1 -15203.653,E2 -15203.653} C_VEL
LIN {X 0,Y 317.754,Z 478.162,A -85,B 0,C 180,E1 -15206.195,E2 -15206.195} C_VEL
LIN {X 0,Y 317.687,Z 479.321,A -85,B 0,C 180,E1 -15208.732,E2 -15208.732} C_VEL
LIN {X 0,Y 317.687,Z 479.318,A -85,B 0,C 180,E1 -15211.268,E2 -15211.268} C_VEL
LIN {X 0,Y 317.755,Z 478.146,A -85,B 0,C 180,E1 -15213.804,E2 -15213.804} C_VEL
LIN {X 0,Y 317.882,Z 475.828,A -85,B 0,C 180,E1 -15216.347,E2 -15216.347} C_VEL
LIN {X 0,Y 318.198,Z 472.313,A -85,B 0,C 180,E1 -15218.894,E2 -15218.894} C_VEL
LIN {X 0,Y 318.768,Z 467.512,A -85,B 0,C 180,E1 -15221.445,E2 -15221.445} C_VEL
LIN {X 0,Y 319.815,Z 461.296,A -85,B 0,C 180,E1 -15223.988,E2 -15223.988} C_VEL
LIN {X 0,Y 321.034,Z 454.574,A -85,B 0,C 180,E1 -15226.208,E2 -15226.208} C_VEL
LIN {X 0,Y 322.672,Z 446.446,A -85,B 0,C 180,E1 -15228.41,E2 -15228.41} C_VEL
LIN {X 0,Y 324.436,Z 438.189,A -85,B 0,C 180,E1 -15230.279,E2 -15230.279} C_VEL
LIN {X 0,Y 326.501,Z 427.491,A -85,B 0,C 180,E1 -15232.32,E2 -15232.32} C_VEL
LIN {X 0,Y 328.852,Z 415.963,A -85,B 0,C 180,E1 -15234.125,E2 -15234.125} C_VEL
LIN {X 0,Y 331.272,Z 403.09,A -85,B 0,C 180,E1 -15235.78,E2 -15235.78} C_VEL
LIN {X 0,Y 333.475,Z 390.339,A -85,B 0,C 180,E1 -15237.113,E2 -15237.113} C_VEL
LIN {X 0,Y 335.638,Z 375.906,A -85,B 0,C 180,E1 -15238.322,E2 -15238.322} C_VEL
LIN {X 0,Y 337.286,Z 362.088,A -85,B 0,C 180,E1 -15239.233,E2 -15239.233} C_VEL
LIN {X 0,Y 338.758,Z 347.433,A -85,B 0,C 180,E1 -15239.948,E2 -15239.948} C_VEL
LIN {X 0,Y 339.804,Z 332.585,A -85,B 0,C 180,E1 -15240.446,E2 -15240.446} C_VEL
LIN {X 0,Y 343.43,Z 220.37,A -85,B 0,C 180,E1 -15242.813,E2 -15242.813} C_VEL
LIN {X 0,Y 343.421,Z 214.371,A -85,B 0,C 180,E1 -15242.96,E2 -15242.96} C_VEL
LIN {X 0,Y 341.987,Z 207.412,A -85,B 0,C 180,E1 -15243.286,E2 -15243.286} C_VEL
LIN {X 0,Y 333.651,Z 188.931,A -85,B 0,C 180,E1 -15244.7,E2 -15244.7} C_VEL
LIN {X 0,Y 326.57,Z 174.956,A -85,B 0,C 180,E1 -15245.933,E2 -15245.933} C_VEL
LIN {X 0,Y 322.887,Z 167.771,A -85,B 0,C 180,E1 -15246.647,E2 -15246.647} C_VEL
LIN {X 0,Y 320.053,Z 158.183,A -85,B 0,C 180,E1 -15249.554,E2 -15249.554} C_VEL
LIN {X 0,Y 319.551,Z 156.339,A -85,B 0,C 180,E1 -15250.244,E2 -15250.244} C_VEL
LIN {X 0,Y 319.521,Z 156.282,A -85,B 0,C 180,E1 -15253.461,E2 -15253.461} C_VEL
LIN {X 0,Y 319.554,Z 156.302,A -85,B 0,C 180,E1 -15257.017,E2 -15257.017} C_VEL
LIN {X 0,Y 319.546,Z 156.272,A -85,B 0,C 180,E1 -15260.371,E2 -15260.371} C_VEL
LIN {X 0,Y 319.559,Z 156.301,A -85,B 0,C 180,E1 -15263.573,E2 -15263.573} C_VEL
LIN {X 0,Y 319.577,Z 156.244,A -85,B 0,C 180,E1 -15266.687,E2 -15266.687} C_VEL
LIN {X 0,Y 319.591,Z 156.281,A -85,B 0,C 180,E1 -15269.617,E2 -15269.617} C_VEL
LIN {X 0,Y 319.61,Z 156.293,A -85,B 0,C 180,E1 -15272.498,E2 -15272.498} C_VEL
LIN {X 0,Y 319.608,Z 156.292,A -85,B 0,C 180,E1 -15275.304,E2 -15275.304} C_VEL
LIN {X 0,Y 319.597,Z 156.287,A -85,B 0,C 180,E1 -15278.048,E2 -15278.048} C_VEL
LIN {X 0,Y 319.69,Z 156.285,A -85,B 0,C 180,E1 -15280.963,E2 -15280.963} C_VEL
LIN {X 0,Y 319.732,Z 156.267,A -85,B 0,C 180,E1 -15285.276,E2 -15285.276} C_VEL
LIN {X 0,Y 319.716,Z 156.277,A -85,B 0,C 180,E1 -15288.59,E2 -15288.59} C_VEL
LIN {X 0,Y 319.858,Z 156.261,A -85,B 0,C 180,E1 -15292.425,E2 -15292.425} C_VEL
LIN {X 0,Y 319.733,Z 156.269,A -85,B 0,C 180,E1 -15294.956,E2 -15294.956} C_VEL
LIN {X 0,Y 319.986,Z 156.235,A -85,B 0,C 180,E1 -15297.483,E2 -15297.483} C_VEL
LIN {X 0,Y 320.113,Z 156.233,A -85,B 0,C 180,E1 -15300,E2 -15300} C_VEL
LIN {X 0,Y 319.963,Z 156.231,A -85,B 0,C 180,E1 -15302.518,E2 -15302.518} C_VEL
LIN {X 0,Y 319.895,Z 156.256,A -85,B 0,C 180,E1 -15306.46,E2 -15306.46} C_VEL
LIN {X 0,Y 319.737,Z 156.273,A -85,B 0,C 180,E1 -15310.128,E2 -15310.128} C_VEL
LIN {X 0,Y 319.732,Z 156.264,A -85,B 0,C 180,E1 -15313.992,E2 -15313.992} C_VEL
LIN {X 0,Y 319.615,Z 156.295,A -85,B 0,C 180,E1 -15317.93,E2 -15317.93} C_VEL
LIN {X 0,Y 319.566,Z 156.3,A -85,B 0,C 180,E1 -15321.955,E2 -15321.955} C_VEL
LIN {X 0,Y 319.553,Z 156.293,A -85,B 0,C 180,E1 -15326.095,E2 -15326.095} C_VEL
LIN {X 0,Y 319.543,Z 156.298,A -85,B 0,C 180,E1 -15328.938,E2 -15328.938} C_VEL
LIN {X 0,Y 319.523,Z 156.249,A -85,B 0,C 180,E1 -15331.863,E2 -15331.863} C_VEL
LIN {X 0,Y 319.58,Z 156.296,A -85,B 0,C 180,E1 -15335.543,E2 -15335.543} C_VEL
LIN {X 0,Y 319.524,Z 156.289,A -85,B 0,C 180,E1 -15338.015,E2 -15338.015} C_VEL
LIN {X 0,Y 319.505,Z 156.277,A -85,B 0,C 180,E1 -15341.593,E2 -15341.593} C_VEL
LIN {X 0,Y 319.487,Z 156.298,A -85,B 0,C 180,E1 -15344.743,E2 -15344.743} C_VEL
LIN {X 0,Y 319.551,Z 156.288,A -85,B 0,C 180,E1 -15347.016,E2 -15347.016} C_VEL
LIN {X 0,Y 319.559,Z 156.462,A -85,B 0,C 180,E1 -15351.085,E2 -15351.085} C_VEL
LIN {X 0,Y 321.539,Z 163.056,A -85,B 0,C 180,E1 -15353.218,E2 -15353.218} C_VEL
LIN {X 0,Y 327.726,Z 174.576,A -85,B 0,C 180,E1 -15354.38,E2 -15354.38} C_VEL
LIN {X 0,Y 336.802,Z 192.818,A -85,B 0,C 180,E1 -15355.944,E2 -15355.944} C_VEL
LIN {X 0,Y 343.72,Z 208.724,A -85,B 0,C 180,E1 -15357.111,E2 -15357.111} C_VEL
LIN {X 0,Y 340.414,Z 313.9,A -85,B 0,C 180,E1 -15359.314,E2 -15359.314} C_VEL
LIN {X 0,Y 339.56,Z 333.056,A -85,B 0,C 180,E1 -15359.788,E2 -15359.788} C_VEL
LIN {X 0,Y 338.379,Z 348.002,A -85,B 0,C 180,E1 -15360.384,E2 -15360.384} C_VEL
LIN {X 0,Y 336.832,Z 363.069,A -85,B 0,C 180,E1 -15361.238,E2 -15361.238} C_VEL
LIN {X 0,Y 335.137,Z 376.271,A -85,B 0,C 180,E1 -15362.213,E2 -15362.213} C_VEL
LIN {X 0,Y 333.121,Z 388.938,A -85,B 0,C 180,E1 -15363.364,E2 -15363.364} C_VEL
LIN {X 0,Y 330.846,Z 402.168,A -85,B 0,C 180,E1 -15364.859,E2 -15364.859} C_VEL
LIN {X 0,Y 328.65,Z 413.24,A -85,B 0,C 180,E1 -15366.362,E2 -15366.362} C_VEL
LIN {X 0,Y 326.499,Z 424.714,A -85,B 0,C 180,E1 -15368.266,E2 -15368.266} C_VEL
LIN {X 0,Y 324.236,Z 435.231,A -85,B 0,C 180,E1 -15370.368,E2 -15370.368} C_VEL
LIN {X 0,Y 322.342,Z 444.227,A -85,B 0,C 180,E1 -15372.555,E2 -15372.555} C_VEL
LIN {X 0,Y 320.82,Z 451.684,A -85,B 0,C 180,E1 -15374.759,E2 -15374.759} C_VEL
LIN {X 0,Y 319.616,Z 458.654,A -85,B 0,C 180,E1 -15377.298,E2 -15377.298} C_VEL
LIN {X 0,Y 318.7,Z 464.133,A -85,B 0,C 180,E1 -15379.839,E2 -15379.839} C_VEL
LIN {X 0,Y 318.125,Z 468.269,A -85,B 0,C 180,E1 -15382.383,E2 -15382.383} C_VEL
LIN {X 0,Y 317.849,Z 471.175,A -85,B 0,C 180,E1 -15384.926,E2 -15384.926} C_VEL
LIN {X 0,Y 317.754,Z 472.923,A -85,B 0,C 180,E1 -15387.465,E2 -15387.465} C_VEL
LIN {X 0,Y 317.703,Z 473.534,A -85,B 0,C 180,E1 -15390,E2 -15390} C_VEL
LIN {X 0,Y 317.754,Z 472.966,A -85,B 0,C 180,E1 -15392.535,E2 -15392.535} C_VEL
LIN {X 0,Y 317.836,Z 471.276,A -85,B 0,C 180,E1 -15395.074,E2 -15395.074} C_VEL
LIN {X 0,Y 318.071,Z 468.424,A -85,B 0,C 180,E1 -15397.618,E2 -15397.618} C_VEL
LIN {X 0,Y 318.657,Z 464.34,A -85,B 0,C 180,E1 -15400.163,E2 -15400.163} C_VEL
LIN {X 0,Y 319.583,Z 458.926,A -85,B 0,C 180,E1 -15402.704,E2 -15402.704} C_VEL
LIN {X 0,Y 320.777,Z 452.031,A -85,B 0,C 180,E1 -15405.243,E2 -15405.243} C_VEL
LIN {X 0,Y 322.55,Z 443.423,A -85,B 0,C 180,E1 -15407.761,E2 -15407.761} C_VEL
LIN {X 0,Y 324.435,Z 434.275,A -85,B 0,C 180,E1 -15409.949,E2 -15409.949} C_VEL
LIN {X 0,Y 326.596,Z 424.306,A -85,B 0,C 180,E1 -15411.918,E2 -15411.918} C_VEL
LIN {X 0,Y 328.826,Z 412.899,A -85,B 0,C 180,E1 -15413.792,E2 -15413.792} C_VEL
LIN {X 0,Y 331.148,Z 400.586,A -85,B 0,C 180,E1 -15415.453,E2 -15415.453} C_VEL
LIN {X 0,Y 333.521,Z 387.001,A -85,B 0,C 180,E1 -15416.94,E2 -15416.94} C_VEL
LIN {X 0,Y 335.607,Z 373.292,A -85,B 0,C 180,E1 -15418.143,E2 -15418.143} C_VEL
LIN {X 0,Y 337.331,Z 358.894,A -85,B 0,C 180,E1 -15419.143,E2 -15419.143} C_VEL
LIN {X 0,Y 338.863,Z 343.383,A -85,B 0,C 180,E1 -15419.938,E2 -15419.938} C_VEL
LIN {X 0,Y 339.93,Z 327.992,A -85,B 0,C 180,E1 -15420.476,E2 -15420.476} C_VEL
LIN {X 0,Y 341.435,Z 284.635,A -85,B 0,C 180,E1 -15421.401,E2 -15421.401} C_VEL
LIN {X 0,Y 341.083,Z 278.834,A -85,B 0,C 180,E1 -15421.578,E2 -15421.578} C_VEL
LIN {X 0,Y 336.817,Z 260.209,A -85,B 0,C 180,E1 -15422.486,E2 -15422.486} C_VEL
LIN {X 0,Y 336.412,Z 254.41,A -85,B 0,C 180,E1 -15422.674,E2 -15422.674} C_VEL
LIN {X 0,Y 337.788,Z 210.816,A -85,B 0,C 180,E1 -15423.608,E2 -15423.608} C_VEL
LIN {X 0,Y 329.871,Z 192.815,A -85,B 0,C 180,E1 -15424.996,E2 -15424.996} C_VEL
LIN {X 0,Y 321.064,Z 175.483,A -85,B 0,C 180,E1 -15426.578,E2 -15426.578} C_VEL
LIN {X 0,Y 314.242,Z 163.14,A -85,B 0,C 180,E1 -15427.908,E2 -15427.908} C_VEL
LIN {X 0,Y 312.492,Z 157.304,A -85,B 0,C 180,E1 -15429.887,E2 -15429.887} C_VEL
LIN {X 0,Y 312.457,Z 157.164,A -85,B 0,C 180,E1 -15433.965,E2 -15433.965} C_VEL
LIN {X 0,Y 312.454,Z 157.168,A -85,B 0,C 180,E1 -15437.925,E2 -15437.925} C_VEL
LIN {X 0,Y 312.477,Z 157.161,A -85,B 0,C 180,E1 -15441.924,E2 -15441.924} C_VEL
LIN {X 0,Y 312.532,Z 157.18,A -85,B 0,C 180,E1 -15444.22,E2 -15444.22} C_VEL
LIN {X 0,Y 312.502,Z 157.124,A -85,B 0,C 180,E1 -15447.333,E2 -15447.333} C_VEL
LIN {X 0,Y 312.507,Z 157.175,A -85,B 0,C 180,E1 -15451.292,E2 -15451.292} C_VEL
LIN {X 0,Y 312.519,Z 157.164,A -85,B 0,C 180,E1 -15454.705,E2 -15454.705} C_VEL
LIN {X 0,Y 312.563,Z 157.175,A -85,B 0,C 180,E1 -15457.527,E2 -15457.527} C_VEL
LIN {X 0,Y 312.565,Z 157.168,A -85,B 0,C 180,E1 -15461.652,E2 -15461.652} C_VEL
LIN {X 0,Y 312.684,Z 157.14,A -85,B 0,C 180,E1 -15465.686,E2 -15465.686} C_VEL
LIN {X 0,Y 312.687,Z 157.154,A -85,B 0,C 180,E1 -15469.641,E2 -15469.641} C_VEL
LIN {X 0,Y 312.802,Z 157.127,A -85,B 0,C 180,E1 -15472.252,E2 -15472.252} C_VEL
LIN {X 0,Y 312.7,Z 157.157,A -85,B 0,C 180,E1 -15474.842,E2 -15474.842} C_VEL
LIN {X 0,Y 312.983,Z 157.107,A -85,B 0,C 180,E1 -15478.713,E2 -15478.713} C_VEL
LIN {X 0,Y 312.984,Z 157.119,A -85,B 0,C 180,E1 -15481.287,E2 -15481.287} C_VEL
LIN {X 0,Y 312.702,Z 157.146,A -85,B 0,C 180,E1 -15485.158,E2 -15485.158} C_VEL
LIN {X 0,Y 312.801,Z 157.139,A -85,B 0,C 180,E1 -15487.747,E2 -15487.747} C_VEL
LIN {X 0,Y 312.666,Z 157.159,A -85,B 0,C 180,E1 -15491.671,E2 -15491.671} C_VEL
LIN {X 0,Y 312.702,Z 157.141,A -85,B 0,C 180,E1 -15494.887,E2 -15494.887} C_VEL
LIN {X 0,Y 312.61,Z 157.165,A -85,B 0,C 180,E1 -15499.225,E2 -15499.225} C_VEL
LIN {X 0,Y 312.527,Z 157.176,A -85,B 0,C 180,E1 -15502.78,E2 -15502.78} C_VEL
LIN {X 0,Y 312.598,Z 157.154,A -85,B 0,C 180,E1 -15505.933,E2 -15505.933} C_VEL
LIN {X 0,Y 312.546,Z 157.17,A -85,B 0,C 180,E1 -15509.65,E2 -15509.65} C_VEL
LIN {X 0,Y 312.52,Z 157.125,A -85,B 0,C 180,E1 -15513.689,E2 -15513.689} C_VEL
LIN {X 0,Y 312.521,Z 157.181,A -85,B 0,C 180,E1 -15517.386,E2 -15517.386} C_VEL
LIN {X 0,Y 312.49,Z 157.146,A -85,B 0,C 180,E1 -15520.709,E2 -15520.709} C_VEL
LIN {X 0,Y 312.452,Z 157.181,A -85,B 0,C 180,E1 -15524.209,E2 -15524.209} C_VEL
LIN {X 0,Y 312.508,Z 157.185,A -85,B 0,C 180,E1 -15528.438,E2 -15528.438} C_VEL
LIN {X 0,Y 312.523,Z 157.371,A -85,B 0,C 180,E1 -15529.03,E2 -15529.03} C_VEL
LIN {X 0,Y 315.629,Z 167.746,A -85,B 0,C 180,E1 -15532.341,E2 -15532.341} C_VEL
LIN {X 0,Y 325.22,Z 185.903,A -85,B 0,C 180,E1 -15534.157,E2 -15534.157} C_VEL
LIN {X 0,Y 332.812,Z 202.086,A -85,B 0,C 180,E1 -15535.51,E2 -15535.51} C_VEL
LIN {X 0,Y 336.728,Z 211.232,A -85,B 0,C 180,E1 -15536.196,E2 -15536.196} C_VEL
LIN {X 0,Y 337.683,Z 217.424,A -85,B 0,C 180,E1 -15536.459,E2 -15536.459} C_VEL
LIN {X 0,Y 334.253,Z 318.598,A -85,B 0,C 180,E1 -15538.597,E2 -15538.597} C_VEL
LIN {X 0,Y 333.439,Z 338.012,A -85,B 0,C 180,E1 -15539.085,E2 -15539.085} C_VEL
LIN {X 0,Y 332.091,Z 353.417,A -85,B 0,C 180,E1 -15539.695,E2 -15539.695} C_VEL
LIN {X 0,Y 330.396,Z 368.271,A -85,B 0,C 180,E1 -15540.534,E2 -15540.534} C_VEL
LIN {X 0,Y 328.465,Z 382.515,A -85,B 0,C 180,E1 -15541.603,E2 -15541.603} C_VEL
LIN {X 0,Y 326.182,Z 396.432,A -85,B 0,C 180,E1 -15542.924,E2 -15542.924} C_VEL
LIN {X 0,Y 323.708,Z 409.331,A -85,B 0,C 180,E1 -15544.437,E2 -15544.437} C_VEL
LIN {X 0,Y 321.288,Z 421.14,A -85,B 0,C 180,E1 -15546.129,E2 -15546.129} C_VEL
LIN {X 0,Y 319.058,Z 431.961,A -85,B 0,C 180,E1 -15548.009,E2 -15548.009} C_VEL
LIN {X 0,Y 317.019,Z 441.138,A -85,B 0,C 180,E1 -15549.902,E2 -15549.902} C_VEL
LIN {X 0,Y 315.129,Z 450.141,A -85,B 0,C 180,E1 -15552.142,E2 -15552.142} C_VEL
LIN {X 0,Y 313.478,Z 458.183,A -85,B 0,C 180,E1 -15554.586,E2 -15554.586} C_VEL
LIN {X 0,Y 312.344,Z 464.573,A -85,B 0,C 180,E1 -15556.997,E2 -15556.997} C_VEL
LIN {X 0,Y 311.429,Z 470.048,A -85,B 0,C 180,E1 -15559.599,E2 -15559.599} C_VEL
LIN {X 0,Y 310.947,Z 474.187,A -85,B 0,C 180,E1 -15562.206,E2 -15562.206} C_VEL
LIN {X 0,Y 310.685,Z 477.087,A -85,B 0,C 180,E1 -15564.808,E2 -15564.808} C_VEL
LIN {X 0,Y 310.644,Z 478.817,A -85,B 0,C 180,E1 -15567.407,E2 -15567.407} C_VEL
LIN {X 0,Y 310.615,Z 479.407,A -85,B 0,C 180,E1 -15570,E2 -15570} C_VEL
LIN {X 0,Y 310.644,Z 478.807,A -85,B 0,C 180,E1 -15572.593,E2 -15572.593} C_VEL
LIN {X 0,Y 310.686,Z 477.065,A -85,B 0,C 180,E1 -15575.191,E2 -15575.191} C_VEL
LIN {X 0,Y 310.948,Z 474.157,A -85,B 0,C 180,E1 -15577.794,E2 -15577.794} C_VEL
LIN {X 0,Y 311.421,Z 470.013,A -85,B 0,C 180,E1 -15580.401,E2 -15580.401} C_VEL
LIN {X 0,Y 312.336,Z 464.523,A -85,B 0,C 180,E1 -15583.004,E2 -15583.004} C_VEL
LIN {X 0,Y 313.553,Z 457.537,A -85,B 0,C 180,E1 -15585.603,E2 -15585.603} C_VEL
LIN {X 0,Y 315.37,Z 448.844,A -85,B 0,C 180,E1 -15588.179,E2 -15588.179} C_VEL
LIN {X 0,Y 317.384,Z 439.608,A -85,B 0,C 180,E1 -15590.412,E2 -15590.412} C_VEL
LIN {X 0,Y 319.241,Z 430.647,A -85,B 0,C 180,E1 -15592.229,E2 -15592.229} C_VEL
LIN {X 0,Y 321.716,Z 419.058,A -85,B 0,C 180,E1 -15594.18,E2 -15594.18} C_VEL
LIN {X 0,Y 324.161,Z 406.83,A -85,B 0,C 180,E1 -15595.869,E2 -15595.869} C_VEL
LIN {X 0,Y 326.647,Z 393.38,A -85,B 0,C 180,E1 -15597.38,E2 -15597.38} C_VEL
LIN {X 0,Y 328.888,Z 379.605,A -85,B 0,C 180,E1 -15598.619,E2 -15598.619} C_VEL
LIN {X 0,Y 330.82,Z 364.568,A -85,B 0,C 180,E1 -15599.687,E2 -15599.687} C_VEL
LIN {X 0,Y 332.467,Z 349.164,A -85,B 0,C 180,E1 -15600.486,E2 -15600.486} C_VEL
LIN {X 0,Y 333.641,Z 333.931,A -85,B 0,C 180,E1 -15601.026,E2 -15601.026} C_VEL
LIN {X 0,Y 337.484,Z 220.575,A -85,B 0,C 180,E1 -15603.459,E2 -15603.459} C_VEL
LIN {X 0,Y 337.456,Z 215.604,A -85,B 0,C 180,E1 -15603.586,E2 -15603.586} C_VEL
LIN {X 0,Y 336.352,Z 210.332,A -85,B 0,C 180,E1 -15603.843,E2 -15603.843} C_VEL
LIN {X 0,Y 328.808,Z 193.421,A -85,B 0,C 180,E1 -15605.167,E2 -15605.167} C_VEL
LIN {X 0,Y 321.499,Z 178.856,A -85,B 0,C 180,E1 -15606.482,E2 -15606.482} C_VEL
LIN {X 0,Y 315.639,Z 167.72,A -85,B 0,C 180,E1 -15607.625,E2 -15607.625} C_VEL
LIN {X 0,Y 312.507,Z 157.314,A -85,B 0,C 180,E1 -15610.968,E2 -15610.968} C_VEL
LIN {X 0,Y 312.451,Z 157.162,A -85,B 0,C 180,E1 -15614.21,E2 -15614.21} C_VEL
LIN {X 0,Y 312.484,Z 157.162,A -85,B 0,C 180,E1 -15617.919,E2 -15617.919} C_VEL
LIN {X 0,Y 312.535,Z 157.17,A -85,B 0,C 180,E1 -15621.911,E2 -15621.911} C_VEL
LIN {X 0,Y 312.506,Z 157.132,A -85,B 0,C 180,E1 -15625.79,E2 -15625.79} C_VEL
LIN {X 0,Y 312.524,Z 157.141,A -85,B 0,C 180,E1 -15628.854,E2 -15628.854} C_VEL
LIN {X 0,Y 312.575,Z 157.173,A -85,B 0,C 180,E1 -15631.825,E2 -15631.825} C_VEL
LIN {X 0,Y 312.587,Z 157.16,A -85,B 0,C 180,E1 -15634.711,E2 -15634.711} C_VEL
LIN {X 0,Y 312.589,Z 157.165,A -85,B 0,C 180,E1 -15637.529,E2 -15637.529} C_VEL
LIN {X 0,Y 312.639,Z 157.166,A -85,B 0,C 180,E1 -15641.657,E2 -15641.657} C_VEL
LIN {X 0,Y 312.695,Z 157.148,A -85,B 0,C 180,E1 -15645.686,E2 -15645.686} C_VEL
LIN {X 0,Y 312.687,Z 157.141,A -85,B 0,C 180,E1 -15649.641,E2 -15649.641} C_VEL
LIN {X 0,Y 312.801,Z 157.139,A -85,B 0,C 180,E1 -15652.253,E2 -15652.253} C_VEL
LIN {X 0,Y 312.702,Z 157.145,A -85,B 0,C 180,E1 -15654.842,E2 -15654.842} C_VEL
LIN {X 0,Y 312.932,Z 157.112,A -85,B 0,C 180,E1 -15657.426,E2 -15657.426} C_VEL
LIN {X 0,Y 313.068,Z 157.111,A -85,B 0,C 180,E1 -15660,E2 -15660} C_VEL
LIN {X 0,Y 312.912,Z 157.109,A -85,B 0,C 180,E1 -15662.575,E2 -15662.575} C_VEL
LIN {X 0,Y 312.85,Z 157.135,A -85,B 0,C 180,E1 -15666.449,E2 -15666.449} C_VEL
LIN {X 0,Y 312.752,Z 157.132,A -85,B 0,C 180,E1 -15669.05,E2 -15669.05} C_VEL
LIN {X 0,Y 312.635,Z 157.159,A -85,B 0,C 180,E1 -15672.991,E2 -15672.991} C_VEL
LIN {X 0,Y 312.622,Z 157.155,A -85,B 0,C 180,E1 -15675.651,E2 -15675.651} C_VEL
LIN {X 0,Y 312.539,Z 157.16,A -85,B 0,C 180,E1 -15679.713,E2 -15679.713} C_VEL
LIN {X 0,Y 312.516,Z 157.181,A -85,B 0,C 180,E1 -15682.776,E2 -15682.776} C_VEL
LIN {X 0,Y 312.487,Z 157.181,A -85,B 0,C 180,E1 -15686.732,E2 -15686.732} C_VEL
LIN {X 0,Y 312.495,Z 157.161,A -85,B 0,C 180,E1 -15689.655,E2 -15689.655} C_VEL
LIN {X 0,Y 312.52,Z 157.132,A -85,B 0,C 180,E1 -15693.689,E2 -15693.689} C_VEL
LIN {X 0,Y 312.511,Z 157.175,A -85,B 0,C 180,E1 -15697.387,E2 -15697.387} C_VEL
LIN {X 0,Y 312.441,Z 157.145,A -85,B 0,C 180,E1 -15700.717,E2 -15700.717} C_VEL
LIN {X 0,Y 312.451,Z 157.183,A -85,B 0,C 180,E1 -15704.21,E2 -15704.21} C_VEL
LIN {X 0,Y 312.455,Z 157.187,A -85,B 0,C 180,E1 -15707.925,E2 -15707.925} C_VEL
LIN {X 0,Y 312.492,Z 157.301,A -85,B 0,C 180,E1 -15710.241,E2 -15710.241} C_VEL
LIN {X 0,Y 314.245,Z 163.093,A -85,B 0,C 180,E1 -15712.209,E2 -15712.209} C_VEL
LIN {X 0,Y 318.65,Z 171.084,A -85,B 0,C 180,E1 -15713.101,E2 -15713.101} C_VEL
LIN {X 0,Y 327.048,Z 187.079,A -85,B 0,C 180,E1 -15714.625,E2 -15714.625} C_VEL
LIN {X 0,Y 335.442,Z 205.19,A -85,B 0,C 180,E1 -15716.099,E2 -15716.099} C_VEL
LIN {X 0,Y 337.715,Z 210.654,A -85,B 0,C 180,E1 -15716.496,E2 -15716.496} C_VEL
LIN {X 0,Y 334.342,Z 313.991,A -85,B 0,C 180,E1 -15718.695,E2 -15718.695} C_VEL
LIN {X 0,Y 333.463,Z 333.138,A -85,B 0,C 180,E1 -15719.176,E2 -15719.176} C_VEL
LIN {X 0,Y 332.224,Z 348.079,A -85,B 0,C 180,E1 -15719.779,E2 -15719.779} C_VEL
LIN {X 0,Y 330.644,Z 362.928,A -85,B 0,C 180,E1 -15720.631,E2 -15720.631} C_VEL
LIN {X 0,Y 328.841,Z 376.541,A -85,B 0,C 180,E1 -15721.653,E2 -15721.653} C_VEL
LIN {X 0,Y 326.547,Z 390.434,A -85,B 0,C 180,E1 -15722.957,E2 -15722.957} C_VEL
LIN {X 0,Y 324.177,Z 403.41,A -85,B 0,C 180,E1 -15724.477,E2 -15724.477} C_VEL
LIN {X 0,Y 321.74,Z 415.259,A -85,B 0,C 180,E1 -15726.165,E2 -15726.165} C_VEL
LIN {X 0,Y 319.58,Z 426.101,A -85,B 0,C 180,E1 -15728.047,E2 -15728.047} C_VEL
LIN {X 0,Y 317.486,Z 435.3,A -85,B 0,C 180,E1 -15729.933,E2 -15729.933} C_VEL
LIN {X 0,Y 315.547,Z 444.296,A -85,B 0,C 180,E1 -15732.167,E2 -15732.167} C_VEL
LIN {X 0,Y 313.923,Z 451.752,A -85,B 0,C 180,E1 -15734.416,E2 -15734.416} C_VEL
LIN {X 0,Y 312.669,Z 458.722,A -85,B 0,C 180,E1 -15737.01,E2 -15737.01} C_VEL
